LIN {X 0,Y 240.088,Z 926.359,A -85,B 0,C 180,E1 -19178.416,E2 -19178.416} C_VEL
LIN {X 0,Y 240.831,Z 922.84,A -85,B 0,C 180,E1 -19181.787,E2 -19181.787} C_VEL
LIN {X 0,Y 242.351,Z 917.839,A -85,B 0,C 180,E1 -19185.129,E2 -19185.129} C_VEL
LIN {X 0,Y 243.941,Z 913.085,A -85,B 0,C 180,E1 -19187.584,E2 -19187.584} C_VEL
LIN {X 0,Y 246.126,Z 906.104,A -85,B 0,C 180,E1 -19190.475,E2 -19190.475} C_VEL
LIN {X 0,Y 249.078,Z 897.538,A -85,B 0,C 180,E1 -19193.267,E2 -19193.267} C_VEL
LIN {X 0,Y 252.071,Z 888.617,A -85,B 0,C 180,E1 -19195.604,E2 -19195.604} C_VEL
LIN {X 0,Y 255.559,Z 877.834,A -85,B 0,C 180,E1 -19197.873,E2 -19197.873} C_VEL
LIN {X 0,Y 258.987,Z 865.759,A -85,B 0,C 180,E1 -19199.91,E2 -19199.91} C_VEL
LIN {X 0,Y 262.112,Z 853.54,A -85,B 0,C 180,E1 -19201.524,E2 -19201.524} C_VEL
LIN {X 0,Y 264.754,Z 841.815,A -85,B 0,C 180,E1 -19202.742,E2 -19202.742} C_VEL
LIN {X 0,Y 267.304,Z 827.813,A -85,B 0,C 180,E1 -19203.853,E2 -19203.853} C_VEL
LIN {X 0,Y 269.3,Z 813.813,A -85,B 0,C 180,E1 -19204.641,E2 -19204.641} C_VEL
LIN {X 0,Y 270.504,Z 800.1,A -85,B 0,C 180,E1 -19205.166,E2 -19205.166} C_VEL
LIN {X 0,Y 273.902,Z 726.368,A -85,B 0,C 180,E1 -19207.051,E2 -19207.051} C_VEL
LIN {X 0,Y 272.415,Z 716.477,A -85,B 0,C 180,E1 -19207.635,E2 -19207.635} C_VEL
LIN {X 0,Y 264.692,Z 699.058,A -85,B 0,C 180,E1 -19209.647,E2 -19209.647} C_VEL
LIN {X 0,Y 256.839,Z 683.886,A -85,B 0,C 180,E1 -19211.794,E2 -19211.794} C_VEL
LIN {X 0,Y 250.877,Z 673.683,A -85,B 0,C 180,E1 -19213.52,E2 -19213.52} C_VEL
LIN {X 0,Y 247.506,Z 668.217,A -85,B 0,C 180,E1 -19214.545,E2 -19214.545} C_VEL
LIN {X 0,Y 244.888,Z 663.741,A -85,B 0,C 180,E1 -19215.408,E2 -19215.408} C_VEL
LIN {X 0,Y 242.509,Z 656.323,A -85,B 0,C 180,E1 -19219.273,E2 -19219.273} C_VEL
LIN {X 0,Y 241.973,Z 654.468,A -85,B 0,C 180,E1 -19220.378,E2 -19220.378} C_VEL
LIN {X 0,Y 242.036,Z 654.449,A -85,B 0,C 180,E1 -19224.498,E2 -19224.498} C_VEL
LIN {X 0,Y 241.976,Z 654.432,A -85,B 0,C 180,E1 -19228.48,E2 -19228.48} C_VEL
LIN {X 0,Y 242.01,Z 654.461,A -85,B 0,C 180,E1 -19232.313,E2 -19232.313} C_VEL
LIN {X 0,Y 242.061,Z 654.455,A -85,B 0,C 180,E1 -19236.017,E2 -19236.017} C_VEL
LIN {X 0,Y 242.039,Z 654.46,A -85,B 0,C 180,E1 -19239.608,E2 -19239.608} C_VEL
LIN {X 0,Y 242.164,Z 654.443,A -85,B 0,C 180,E1 -19243.279,E2 -19243.279} C_VEL
LIN {X 0,Y 242.182,Z 654.444,A -85,B 0,C 180,E1 -19248.28,E2 -19248.28} C_VEL
LIN {X 0,Y 242.401,Z 654.404,A -85,B 0,C 180,E1 -19251.665,E2 -19251.665} C_VEL
LIN {X 0,Y 242.258,Z 654.422,A -85,B 0,C 180,E1 -19255.008,E2 -19255.008} C_VEL
LIN {X 0,Y 242.637,Z 654.387,A -85,B 0,C 180,E1 -19258.341,E2 -19258.341} C_VEL
LIN {X 0,Y 242.637,Z 654.377,A -85,B 0,C 180,E1 -19261.66,E2 -19261.66} C_VEL
LIN {X 0,Y 242.423,Z 654.403,A -85,B 0,C 180,E1 -19266.684,E2 -19266.684} C_VEL
LIN {X 0,Y 242.269,Z 654.42,A -85,B 0,C 180,E1 -19270.024,E2 -19270.024} C_VEL
LIN {X 0,Y 242.169,Z 654.432,A -85,B 0,C 180,E1 -19275.141,E2 -19275.141} C_VEL
LIN {X 0,Y 242.073,Z 654.448,A -85,B 0,C 180,E1 -19278.625,E2 -19278.625} C_VEL
LIN {X 0,Y 242.007,Z 654.463,A -85,B 0,C 180,E1 -19282.181,E2 -19282.181} C_VEL
LIN {X 0,Y 242.034,Z 654.461,A -85,B 0,C 180,E1 -19285.822,E2 -19285.822} C_VEL
LIN {X 0,Y 241.971,Z 654.433,A -85,B 0,C 180,E1 -19289.589,E2 -19289.589} C_VEL
LIN {X 0,Y 241.981,Z 654.462,A -85,B 0,C 180,E1 -19293.493,E2 -19293.493} C_VEL
LIN {X 0,Y 241.984,Z 654.464,A -85,B 0,C 180,E1 -19297.584,E2 -19297.584} C_VEL
LIN {X 0,Y 241.941,Z 654.466,A -85,B 0,C 180,E1 -19299.017,E2 -19299.017} C_VEL
LIN {X 0,Y 242.888,Z 657.248,A -85,B 0,C 180,E1 -19299.397,E2 -19299.397} C_VEL
LIN {X 0,Y 245.069,Z 659.506,A -85,B 0,C 180,E1 -19300.06,E2 -19300.06} C_VEL
LIN {X 0,Y 247.535,Z 663.319,A -85,B 0,C 180,E1 -19300.837,E2 -19300.837} C_VEL
LIN {X 0,Y 248.885,Z 665.08,A -85,B 0,C 180,E1 -19301.238,E2 -19301.238} C_VEL
LIN {X 0,Y 252.713,Z 670.642,A -85,B 0,C 180,E1 -19302.36,E2 -19302.36} C_VEL
LIN {X 0,Y 259.191,Z 680.306,A -85,B 0,C 180,E1 -19304.146,E2 -19304.146} C_VEL
LIN {X 0,Y 265.13,Z 690.246,A -85,B 0,C 180,E1 -19305.702,E2 -19305.702} C_VEL
LIN {X 0,Y 272.196,Z 704.465,A -85,B 0,C 180,E1 -19307.5,E2 -19307.5} C_VEL
LIN {X 0,Y 274.562,Z 709.751,A -85,B 0,C 180,E1 -19308.089,E2 -19308.089} C_VEL
LIN {X 0,Y 271.055,Z 786.527,A -85,B 0,C 180,E1 -19310.079,E2 -19310.079} C_VEL
LIN {X 0,Y 269.646,Z 801.309,A -85,B 0,C 180,E1 -19310.739,E2 -19310.739} C_VEL
LIN {X 0,Y 267.76,Z 814.787,A -85,B 0,C 180,E1 -19311.617,E2 -19311.617} C_VEL
LIN {X 0,Y 265.371,Z 827.421,A -85,B 0,C 180,E1 -19312.703,E2 -19312.703} C_VEL
LIN {X 0,Y 262.585,Z 840.272,A -85,B 0,C 180,E1 -19314.163,E2 -19314.163} C_VEL
LIN {X 0,Y 259.624,Z 851.868,A -85,B 0,C 180,E1 -19315.827,E2 -19315.827} C_VEL
LIN {X 0,Y 256.55,Z 862.473,A -85,B 0,C 180,E1 -19317.711,E2 -19317.711} C_VEL
LIN {X 0,Y 253.359,Z 872.972,A -85,B 0,C 180,E1 -19320.046,E2 -19320.046} C_VEL
LIN {X 0,Y 250.379,Z 881.602,A -85,B 0,C 180,E1 -19322.41,E2 -19322.41} C_VEL
LIN {X 0,Y 247.78,Z 888.746,A -85,B 0,C 180,E1 -19324.82,E2 -19324.82} C_VEL
LIN {X 0,Y 245.672,Z 894.661,A -85,B 0,C 180,E1 -19327.282,E2 -19327.282} C_VEL
LIN {X 0,Y 243.34,Z 900.946,A -85,B 0,C 180,E1 -19330.602,E2 -19330.602} C_VEL
LIN {X 0,Y 241.933,Z 904.957,A -85,B 0,C 180,E1 -19333.464,E2 -19333.464} C_VEL
LIN {X 0,Y 240.798,Z 908.016,A -85,B 0,C 180,E1 -19336.498,E2 -19336.498} C_VEL
LIN {X 0,Y 240.149,Z 910.096,A -85,B 0,C 180,E1 -19339.887,E2 -19339.887} C_VEL
LIN {X 0,Y 239.958,Z 910.837,A -85,B 0,C 180,E1 -19343.272,E2 -19343.272} C_VEL
LIN {X 0,Y 239.916,Z 910.27,A -85,B 0,C 180,E1 -19346.641,E2 -19346.641} C_VEL
LIN {X 0,Y 240.051,Z 908.394,A -85,B 0,C 180,E1 -19350,E2 -19350} C_VEL
LIN {X 0,Y 240.514,Z 905.147,A -85,B 0,C 180,E1 -19353.351,E2 -19353.351} C_VEL
LIN {X 0,Y 241.617,Z 900.424,A -85,B 0,C 180,E1 -19356.682,E2 -19356.682} C_VEL
LIN {X 0,Y 242.775,Z 895.871,A -85,B 0,C 180,E1 -19359.162,E2 -19359.162} C_VEL
LIN {X 0,Y 244.53,Z 889.16,A -85,B 0,C 180,E1 -19362.063,E2 -19362.063} C_VEL
LIN {X 0,Y 246.44,Z 881.04,A -85,B 0,C 180,E1 -19364.872,E2 -19364.872} C_VEL
LIN {X 0,Y 248.908,Z 872.445,A -85,B 0,C 180,E1 -19367.246,E2 -19367.246} C_VEL
LIN {X 0,Y 251.545,Z 862.05,A -85,B 0,C 180,E1 -19369.589,E2 -19369.589} C_VEL
LIN {X 0,Y 254.179,Z 850.427,A -85,B 0,C 180,E1 -19371.705,E2 -19371.705} C_VEL
LIN {X 0,Y 256.478,Z 838.788,A -85,B 0,C 180,E1 -19373.412,E2 -19373.412} C_VEL
LIN {X 0,Y 258.792,Z 825.949,A -85,B 0,C 180,E1 -19374.894,E2 -19374.894} C_VEL
LIN {X 0,Y 260.773,Z 812.564,A -85,B 0,C 180,E1 -19376.081,E2 -19376.081} C_VEL
LIN {X 0,Y 262.277,Z 798.574,A -85,B 0,C 180,E1 -19376.992,E2 -19376.992} C_VEL
LIN {X 0,Y 263.296,Z 784.338,A -85,B 0,C 180,E1 -19377.607,E2 -19377.607} C_VEL
LIN {X 0,Y 266.607,Z 702.616,A -85,B 0,C 180,E1 -19379.747,E2 -19379.747} C_VEL
LIN {X 0,Y 259.944,Z 686.637,A -85,B 0,C 180,E1 -19381.221,E2 -19381.221} C_VEL
LIN {X 0,Y 254.009,Z 675.196,A -85,B 0,C 180,E1 -19382.527,E2 -19382.527} C_VEL
LIN {X 0,Y 245.648,Z 661.352,A -85,B 0,C 180,E1 -19384.431,E2 -19384.431} C_VEL
LIN {X 0,Y 243.844,Z 658.424,A -85,B 0,C 180,E1 -19384.864,E2 -19384.864} C_VEL
LIN {X 0,Y 242.334,Z 655.911,A -85,B 0,C 180,E1 -19385.235,E2 -19385.235} C_VEL
LIN {X 0,Y 242,Z 654.467,A -85,B 0,C 180,E1 -19385.38,E2 -19385.38} C_VEL
LIN {X 0,Y 241.936,Z 654.453,A -85,B 0,C 180,E1 -19389.723,E2 -19389.723} C_VEL
LIN {X 0,Y 241.919,Z 654.469,A -85,B 0,C 180,E1 -19394.205,E2 -19394.205} C_VEL
LIN {X 0,Y 241.911,Z 654.475,A -85,B 0,C 180,E1 -19398.071,E2 -19398.071} C_VEL
LIN {X 0,Y 241.967,Z 654.433,A -85,B 0,C 180,E1 -19402.413,E2 -19402.413} C_VEL
LIN {X 0,Y 241.982,Z 654.466,A -85,B 0,C 180,E1 -19406.507,E2 -19406.507} C_VEL
LIN {X 0,Y 241.98,Z 654.454,A -85,B 0,C 180,E1 -19410.612,E2 -19410.612} C_VEL
LIN {X 0,Y 242.035,Z 654.455,A -85,B 0,C 180,E1 -19414.179,E2 -19414.179} C_VEL
LIN {X 0,Y 242.025,Z 654.46,A -85,B 0,C 180,E1 -19418.315,E2 -19418.315} C_VEL
LIN {X 0,Y 242.118,Z 654.43,A -85,B 0,C 180,E1 -19423.316,E2 -19423.316} C_VEL
LIN {X 0,Y 242.17,Z 654.43,A -85,B 0,C 180,E1 -19428.278,E2 -19428.278} C_VEL
LIN {X 0,Y 242.388,Z 654.408,A -85,B 0,C 180,E1 -19431.664,E2 -19431.664} C_VEL
LIN {X 0,Y 242.242,Z 654.429,A -85,B 0,C 180,E1 -19435.006,E2 -19435.006} C_VEL
LIN {X 0,Y 242.636,Z 654.386,A -85,B 0,C 180,E1 -19438.34,E2 -19438.34} C_VEL
LIN {X 0,Y 242.592,Z 654.382,A -85,B 0,C 180,E1 -19441.872,E2 -19441.872} C_VEL
LIN {X 0,Y 241.73,Z 654.5,A -85,B 0,C 180,E1 -19443.255,E2 -19443.255} C_VEL
LIN {X 0,Y 238.797,Z 654.862,A -85,B 0,C 180,E1 -19445.512,E2 -19445.512} C_VEL
LIN {X 0,Y 236.412,Z 655.16,A -85,B 0,C 180,E1 -19447.35,E2 -19447.35} C_VEL
LIN {X 0,Y 235.388,Z 655.288,A -85,B 0,C 180,E1 -19448.776,E2 -19448.776} C_VEL
LIN {X 0,Y 235.297,Z 655.295,A -85,B 0,C 180,E1 -19449.259,E2 -19449.259} C_VEL
LIN {X 0,Y 235.109,Z 655.321,A -85,B 0,C 180,E1 -19453.835,E2 -19453.835} C_VEL
LIN {X 0,Y 235.07,Z 655.326,A -85,B 0,C 180,E1 -19457.396,E2 -19457.396} C_VEL
LIN {X 0,Y 234.979,Z 655.338,A -85,B 0,C 180,E1 -19462,E2 -19462} C_VEL
LIN {X 0,Y 234.97,Z 655.334,A -85,B 0,C 180,E1 -19466.657,E2 -19466.657} C_VEL
LIN {X 0,Y 234.934,Z 655.34,A -85,B 0,C 180,E1 -19470.567,E2 -19470.567} C_VEL
LIN {X 0,Y 234.962,Z 655.339,A -85,B 0,C 180,E1 -19474.632,E2 -19474.632} C_VEL
LIN {X 0,Y 234.968,Z 655.339,A -85,B 0,C 180,E1 -19478.952,E2 -19478.952} C_VEL
LIN {X 0,Y 234.949,Z 655.341,A -85,B 0,C 180,E1 -19483.471,E2 -19483.471} C_VEL
LIN {X 0,Y 234.953,Z 655.525,A -85,B 0,C 180,E1 -19484.67,E2 -19484.67} C_VEL
LIN {X 0,Y 237.458,Z 664.503,A -85,B 0,C 180,E1 -19488.654,E2 -19488.654} C_VEL
LIN {X 0,Y 244.776,Z 678.336,A -85,B 0,C 180,E1 -19490.52,E2 -19490.52} C_VEL
LIN {X 0,Y 252.132,Z 694.464,A -85,B 0,C 180,E1 -19492.323,E2 -19492.323} C_VEL
LIN {X 0,Y 257.755,Z 708.307,A -85,B 0,C 180,E1 -19493.657,E2 -19493.657} C_VEL
LIN {X 0,Y 259.899,Z 725.152,A -85,B 0,C 180,E1 -19494.519,E2 -19494.519} C_VEL
LIN {X 0,Y 256.62,Z 803.382,A -85,B 0,C 180,E1 -19496.625,E2 -19496.625} C_VEL
LIN {X 0,Y 255.268,Z 817.931,A -85,B 0,C 180,E1 -19497.295,E2 -19497.295} C_VEL
LIN {X 0,Y 253.467,Z 831.442,A -85,B 0,C 180,E1 -19498.209,E2 -19498.209} C_VEL
LIN {X 0,Y 251.375,Z 843.741,A -85,B 0,C 180,E1 -19499.32,E2 -19499.32} C_VEL
LIN {X 0,Y 248.825,Z 856.669,A -85,B 0,C 180,E1 -19500.842,E2 -19500.842} C_VEL
LIN {X 0,Y 246.309,Z 868.123,A -85,B 0,C 180,E1 -19502.549,E2 -19502.549} C_VEL
LIN {X 0,Y 243.841,Z 878.189,A -85,B 0,C 180,E1 -19504.384,E2 -19504.384} C_VEL
LIN {X 0,Y 241.346,Z 887.356,A -85,B 0,C 180,E1 -19506.397,E2 -19506.397} C_VEL
LIN {X 0,Y 238.958,Z 896.569,A -85,B 0,C 180,E1 -19508.882,E2 -19508.882} C_VEL
LIN {X 0,Y 236.842,Z 904.466,A -85,B 0,C 180,E1 -19511.489,E2 -19511.489} C_VEL
LIN {X 0,Y 235.207,Z 911.563,A -85,B 0,C 180,E1 -19514.4,E2 -19514.4} C_VEL
LIN {X 0,Y 234.076,Z 916.69,A -85,B 0,C 180,E1 -19516.986,E2 -19516.986} C_VEL
LIN {X 0,Y 233.168,Z 921.968,A -85,B 0,C 180,E1 -19520.457,E2 -19520.457} C_VEL
LIN {X 0,Y 232.856,Z 924.929,A -85,B 0,C 180,E1 -19523.066,E2 -19523.066} C_VEL
LIN {X 0,Y 232.831,Z 926.555,A -85,B 0,C 180,E1 -19524.939,E2 -19524.939} C_VEL
LIN {X 0,Y 232.827,Z 928.419,A -85,B 0,C 180,E1 -19528.27,E2 -19528.27} C_VEL
LIN {X 0,Y 232.888,Z 928.888,A -85,B 0,C 180,E1 -19530,E2 -19530} C_VEL
LIN {X 0,Y 232.816,Z 929.01,A -85,B 0,C 180,E1 -19531.73,E2 -19531.73} C_VEL
LIN {X 0,Y 232.742,Z 928.246,A -85,B 0,C 180,E1 -19535.197,E2 -19535.197} C_VEL
LIN {X 0,Y 233.039,Z 926.14,A -85,B 0,C 180,E1 -19538.673,E2 -19538.673} C_VEL
LIN {X 0,Y 233.826,Z 922.646,A -85,B 0,C 180,E1 -19542.145,E2 -19542.145} C_VEL
LIN {X 0,Y 235.44,Z 917.672,A -85,B 0,C 180,E1 -19545.584,E2 -19545.584} C_VEL
LIN {X 0,Y 237.262,Z 912.366,A -85,B 0,C 180,E1 -19548.38,E2 -19548.38} C_VEL
LIN {X 0,Y 239.846,Z 904.878,A -85,B 0,C 180,E1 -19551.486,E2 -19551.486} C_VEL
LIN {X 0,Y 243.033,Z 896.111,A -85,B 0,C 180,E1 -19554.335,E2 -19554.335} C_VEL
LIN {X 0,Y 246.281,Z 886.961,A -85,B 0,C 180,E1 -19556.708,E2 -19556.708} C_VEL
LIN {X 0,Y 249.773,Z 876.499,A -85,B 0,C 180,E1 -19558.897,E2 -19558.897} C_VEL
LIN {X 0,Y 252.838,Z 865.845,A -85,B 0,C 180,E1 -19560.714,E2 -19560.714} C_VEL
LIN {X 0,Y 256.085,Z 853.738,A -85,B 0,C 180,E1 -19562.354,E2 -19562.354} C_VEL
LIN {X 0,Y 258.826,Z 842.104,A -85,B 0,C 180,E1 -19563.59,E2 -19563.59} C_VEL
LIN {X 0,Y 261.467,Z 828.337,A -85,B 0,C 180,E1 -19564.715,E2 -19564.715} C_VEL
LIN {X 0,Y 263.632,Z 813.751,A -85,B 0,C 180,E1 -19565.555,E2 -19565.555} C_VEL
LIN {X 0,Y 264.913,Z 799.46,A -85,B 0,C 180,E1 -19566.11,E2 -19566.11} C_VEL
LIN {X 0,Y 268.353,Z 727.432,A -85,B 0,C 180,E1 -19567.979,E2 -19567.979} C_VEL
LIN {X 0,Y 267.061,Z 719.125,A -85,B 0,C 180,E1 -19568.499,E2 -19568.499} C_VEL
LIN {X 0,Y 259.143,Z 701.17,A -85,B 0,C 180,E1 -19570.667,E2 -19570.667} C_VEL
LIN {X 0,Y 251.705,Z 687.021,A -85,B 0,C 180,E1 -19572.8,E2 -19572.8} C_VEL
LIN {X 0,Y 246.944,Z 678.673,A -85,B 0,C 180,E1 -19574.25,E2 -19574.25} C_VEL
LIN {X 0,Y 240.455,Z 668.201,A -85,B 0,C 180,E1 -19576.349,E2 -19576.349} C_VEL
LIN {X 0,Y 237.454,Z 663.229,A -85,B 0,C 180,E1 -19577.462,E2 -19577.462} C_VEL
LIN {X 0,Y 234.985,Z 655.315,A -85,B 0,C 180,E1 -19581.981,E2 -19581.981} C_VEL
LIN {X 0,Y 234.95,Z 655.32,A -85,B 0,C 180,E1 -19586.883,E2 -19586.883} C_VEL
LIN {X 0,Y 234.954,Z 655.339,A -85,B 0,C 180,E1 -19591.407,E2 -19591.407} C_VEL
LIN {X 0,Y 234.99,Z 655.336,A -85,B 0,C 180,E1 -19595.247,E2 -19595.247} C_VEL
LIN {X 0,Y 235.012,Z 655.332,A -85,B 0,C 180,E1 -19598.97,E2 -19598.97} C_VEL
LIN {X 0,Y 235.097,Z 655.32,A -85,B 0,C 180,E1 -19603.06,E2 -19603.06} C_VEL
LIN {X 0,Y 235.115,Z 655.32,A -85,B 0,C 180,E1 -19607.923,E2 -19607.923} C_VEL
LIN {X 0,Y 235.332,Z 655.283,A -85,B 0,C 180,E1 -19611.413,E2 -19611.413} C_VEL
LIN {X 0,Y 235.394,Z 655.289,A -85,B 0,C 180,E1 -19613.142,E2 -19613.142} C_VEL
LIN {X 0,Y 235.597,Z 655.265,A -85,B 0,C 180,E1 -19618.291,E2 -19618.291} C_VEL
LIN {X 0,Y 235.597,Z 655.254,A -85,B 0,C 180,E1 -19621.71,E2 -19621.71} C_VEL
LIN {X 0,Y 235.375,Z 655.283,A -85,B 0,C 180,E1 -19626.86,E2 -19626.86} C_VEL
LIN {X 0,Y 235.216,Z 655.297,A -85,B 0,C 180,E1 -19630.328,E2 -19630.328} C_VEL
LIN {X 0,Y 235.115,Z 655.312,A -85,B 0,C 180,E1 -19635.607,E2 -19635.607} C_VEL
LIN {X 0,Y 235.009,Z 655.325,A -85,B 0,C 180,E1 -19639.206,E2 -19639.206} C_VEL
LIN {X 0,Y 234.952,Z 655.335,A -85,B 0,C 180,E1 -19642.884,E2 -19642.884} C_VEL
LIN {X 0,Y 234.948,Z 655.332,A -85,B 0,C 180,E1 -19646.661,E2 -19646.661} C_VEL
LIN {X 0,Y 234.901,Z 655.321,A -85,B 0,C 180,E1 -19650.573,E2 -19650.573} C_VEL
LIN {X 0,Y 234.927,Z 655.341,A -85,B 0,C 180,E1 -19654.639,E2 -19654.639} C_VEL
LIN {X 0,Y 234.918,Z 655.376,A -85,B 0,C 180,E1 -19657.087,E2 -19657.087} C_VEL
LIN {X 0,Y 235.79,Z 657.948,A -85,B 0,C 180,E1 -19657.463,E2 -19657.463} C_VEL
LIN {X 0,Y 237.848,Z 660.234,A -85,B 0,C 180,E1 -19658.157,E2 -19658.157} C_VEL
LIN {X 0,Y 238.51,Z 661.013,A -85,B 0,C 180,E1 -19658.377,E2 -19658.377} C_VEL
LIN {X 0,Y 240.624,Z 664.296,A -85,B 0,C 180,E1 -19659.102,E2 -19659.102} C_VEL
LIN {X 0,Y 242.07,Z 666.019,A -85,B 0,C 180,E1 -19659.563,E2 -19659.563} C_VEL
LIN {X 0,Y 250.555,Z 678.145,A -85,B 0,C 180,E1 -19662.162,E2 -19662.162} C_VEL
LIN {X 0,Y 259.292,Z 692.068,A -85,B 0,C 180,E1 -19664.605,E2 -19664.605} C_VEL
LIN {X 0,Y 267.106,Z 707.667,A -85,B 0,C 180,E1 -19666.69,E2 -19666.69} C_VEL
LIN {X 0,Y 268.933,Z 711.817,A -85,B 0,C 180,E1 -19667.168,E2 -19667.168} C_VEL
LIN {X 0,Y 267.067,Z 753.218,A -85,B 0,C 180,E1 -19668.251,E2 -19668.251} C_VEL
LIN {X 0,Y 265.399,Z 787.321,A -85,B 0,C 180,E1 -19669.175,E2 -19669.175} C_VEL
LIN {X 0,Y 263.941,Z 801.924,A -85,B 0,C 180,E1 -19669.844,E2 -19669.844} C_VEL
LIN {X 0,Y 261.893,Z 815.882,A -85,B 0,C 180,E1 -19670.779,E2 -19670.779} C_VEL
LIN {X 0,Y 259.484,Z 828.085,A -85,B 0,C 180,E1 -19671.857,E2 -19671.857} C_VEL
LIN {X 0,Y 256.459,Z 841.42,A -85,B 0,C 180,E1 -19673.414,E2 -19673.414} C_VEL
LIN {X 0,Y 253.39,Z 852.858,A -85,B 0,C 180,E1 -19675.107,E2 -19675.107} C_VEL
LIN {X 0,Y 250.494,Z 862.361,A -85,B 0,C 180,E1 -19676.832,E2 -19676.832} C_VEL
LIN {X 0,Y 247.159,Z 872.924,A -85,B 0,C 180,E1 -19679.214,E2 -19679.214} C_VEL
LIN {X 0,Y 244.011,Z 881.608,A -85,B 0,C 180,E1 -19681.626,E2 -19681.626} C_VEL
LIN {X 0,Y 240.87,Z 889.951,A -85,B 0,C 180,E1 -19684.53,E2 -19684.53} C_VEL
LIN {X 0,Y 238.345,Z 896.529,A -85,B 0,C 180,E1 -19687.46,E2 -19687.46} C_VEL
LIN {X 0,Y 236.048,Z 902.381,A -85,B 0,C 180,E1 -19690.882,E2 -19690.882} C_VEL
LIN {X 0,Y 234.444,Z 906.642,A -85,B 0,C 180,E1 -19694.348,E2 -19694.348} C_VEL
LIN {X 0,Y 233.344,Z 909.448,A -85,B 0,C 180,E1 -19697.829,E2 -19697.829} C_VEL
LIN {X 0,Y 232.919,Z 910.883,A -85,B 0,C 180,E1 -19701.323,E2 -19701.323} C_VEL
LIN {X 0,Y 232.848,Z 910.997,A -85,B 0,C 180,E1 -19704.805,E2 -19704.805} C_VEL
LIN {X 0,Y 232.898,Z 909.81,A -85,B 0,C 180,E1 -19708.271,E2 -19708.271} C_VEL
LIN {X 0,Y 233.148,Z 907.301,A -85,B 0,C 180,E1 -19711.728,E2 -19711.728} C_VEL
LIN {X 0,Y 233.95,Z 903.37,A -85,B 0,C 180,E1 -19715.171,E2 -19715.171} C_VEL
LIN {X 0,Y 235.4,Z 897.898,A -85,B 0,C 180,E1 -19718.585,E2 -19718.585} C_VEL
LIN {X 0,Y 236.816,Z 892.722,A -85,B 0,C 180,E1 -19721.122,E2 -19721.122} C_VEL
LIN {X 0,Y 238.671,Z 885.274,A -85,B 0,C 180,E1 -19724.06,E2 -19724.06} C_VEL
LIN {X 0,Y 240.88,Z 877.503,A -85,B 0,C 180,E1 -19726.527,E2 -19726.527} C_VEL
LIN {X 0,Y 243.5,Z 868.124,A -85,B 0,C 180,E1 -19728.948,E2 -19728.948} C_VEL
LIN {X 0,Y 246.133,Z 857.752,A -85,B 0,C 180,E1 -19731.131,E2 -19731.131} C_VEL
LIN {X 0,Y 248.41,Z 847.594,A -85,B 0,C 180,E1 -19732.893,E2 -19732.893} C_VEL
LIN {X 0,Y 250.613,Z 836.757,A -85,B 0,C 180,E1 -19734.434,E2 -19734.434} C_VEL
LIN {X 0,Y 252.718,Z 825.153,A -85,B 0,C 180,E1 -19735.755,E2 -19735.755} C_VEL
LIN {X 0,Y 254.793,Z 811.326,A -85,B 0,C 180,E1 -19736.962,E2 -19736.962} C_VEL
LIN {X 0,Y 256.248,Z 797.577,A -85,B 0,C 180,E1 -19737.846,E2 -19737.846} C_VEL
LIN {X 0,Y 257.269,Z 783.689,A -85,B 0,C 180,E1 -19738.433,E2 -19738.433} C_VEL
LIN {X 0,Y 260.523,Z 704.324,A -85,B 0,C 180,E1 -19740.558,E2 -19740.558} C_VEL
LIN {X 0,Y 253.921,Z 688.54,A -85,B 0,C 180,E1 -19742.087,E2 -19742.087} C_VEL
LIN {X 0,Y 246.236,Z 674.417,A -85,B 0,C 180,E1 -19743.858,E2 -19743.858} C_VEL
LIN {X 0,Y 238.878,Z 662.529,A -85,B 0,C 180,E1 -19745.641,E2 -19745.641} C_VEL
LIN {X 0,Y 237.106,Z 659.66,A -85,B 0,C 180,E1 -19746.094,E2 -19746.094} C_VEL
LIN {X 0,Y 235.318,Z 657.035,A -85,B 0,C 180,E1 -19746.55,E2 -19746.55} C_VEL
LIN {X 0,Y 234.909,Z 655.347,A -85,B 0,C 180,E1 -19746.753,E2 -19746.753} C_VEL
LIN {X 0,Y 234.915,Z 655.332,A -85,B 0,C 180,E1 -19748.935,E2 -19748.935} C_VEL
LIN {X 0,Y 234.878,Z 655.347,A -85,B 0,C 180,E1 -19753.489,E2 -19753.489} C_VEL
LIN {X 0,Y 234.865,Z 655.35,A -85,B 0,C 180,E1 -19756.508,E2 -19756.508} C_VEL
LIN {X 0,Y 234.92,Z 655.323,A -85,B 0,C 180,E1 -19761.078,E2 -19761.078} C_VEL
LIN {X 0,Y 234.924,Z 655.335,A -85,B 0,C 180,E1 -19765.36,E2 -19765.36} C_VEL
LIN {X 0,Y 234.902,Z 655.333,A -85,B 0,C 180,E1 -19769.427,E2 -19769.427} C_VEL
LIN {X 0,Y 234.971,Z 655.336,A -85,B 0,C 180,E1 -19773.806,E2 -19773.806} C_VEL
LIN {X 0,Y 234.992,Z 655.338,A -85,B 0,C 180,E1 -19778.967,E2 -19778.967} C_VEL
LIN {X 0,Y 235.059,Z 655.307,A -85,B 0,C 180,E1 -19783.092,E2 -19783.092} C_VEL
LIN {X 0,Y 235.102,Z 655.313,A -85,B 0,C 180,E1 -19787.921,E2 -19787.921} C_VEL
LIN {X 0,Y 235.322,Z 655.286,A -85,B 0,C 180,E1 -19791.412,E2 -19791.412} C_VEL
LIN {X 0,Y 235.358,Z 655.292,A -85,B 0,C 180,E1 -19793.139,E2 -19793.139} C_VEL
LIN {X 0,Y 235.595,Z 655.263,A -85,B 0,C 180,E1 -19798.29,E2 -19798.29} C_VEL
LIN {X 0,Y 235.581,Z 655.256,A -85,B 0,C 180,E1 -19801.781,E2 -19801.781} C_VEL
LIN {X 0,Y 235.375,Z 655.285,A -85,B 0,C 180,E1 -19806.859,E2 -19806.859} C_VEL
LIN {X 0,Y 235.297,Z 655.295,A -85,B 0,C 180,E1 -19809.259,E2 -19809.259} C_VEL
LIN {X 0,Y 234.588,Z 655.383,A -85,B 0,C 180,E1 -19810.687,E2 -19810.687} C_VEL
LIN {X 0,Y 231.655,Z 655.753,A -85,B 0,C 180,E1 -19813.013,E2 -19813.013} C_VEL
LIN {X 0,Y 229.179,Z 656.054,A -85,B 0,C 180,E1 -19814.91,E2 -19814.91} C_VEL
LIN {X 0,Y 228.12,Z 656.187,A -85,B 0,C 180,E1 -19816.385,E2 -19816.385} C_VEL
LIN {X 0,Y 228.035,Z 656.199,A -85,B 0,C 180,E1 -19816.885,E2 -19816.885} C_VEL
LIN {X 0,Y 227.949,Z 656.213,A -85,B 0,C 180,E1 -19821.714,E2 -19821.714} C_VEL
LIN {X 0,Y 227.944,Z 656.21,A -85,B 0,C 180,E1 -19826.602,E2 -19826.602} C_VEL
LIN {X 0,Y 227.91,Z 656.215,A -85,B 0,C 180,E1 -19830.296,E2 -19830.296} C_VEL
LIN {X 0,Y 227.891,Z 656.219,A -85,B 0,C 180,E1 -19833.718,E2 -19833.718} C_VEL
LIN {X 0,Y 227.872,Z 656.226,A -85,B 0,C 180,E1 -19838.085,E2 -19838.085} C_VEL
LIN {X 0,Y 227.895,Z 656.221,A -85,B 0,C 180,E1 -19842.722,E2 -19842.722} C_VEL
LIN {X 0,Y 227.914,Z 656.299,A -85,B 0,C 180,E1 -19843.474,E2 -19843.474} C_VEL
LIN {X 0,Y 230.089,Z 664.076,A -85,B 0,C 180,E1 -19847.144,E2 -19847.144} C_VEL
LIN {X 0,Y 232.529,Z 668.575,A -85,B 0,C 180,E1 -19847.83,E2 -19847.83} C_VEL
LIN {X 0,Y 238.864,Z 680.448,A -85,B 0,C 180,E1 -19849.524,E2 -19849.524} C_VEL
LIN {X 0,Y 246.196,Z 696.303,A -85,B 0,C 180,E1 -19851.407,E2 -19851.407} C_VEL
LIN {X 0,Y 252.056,Z 710.872,A -85,B 0,C 180,E1 -19852.87,E2 -19852.87} C_VEL
LIN {X 0,Y 253.95,Z 726.459,A -85,B 0,C 180,E1 -19853.686,E2 -19853.686} C_VEL
LIN {X 0,Y 250.594,Z 802.921,A -85,B 0,C 180,E1 -19855.778,E2 -19855.778} C_VEL
LIN {X 0,Y 249.212,Z 817.485,A -85,B 0,C 180,E1 -19856.457,E2 -19856.457} C_VEL
LIN {X 0,Y 247.489,Z 830.481,A -85,B 0,C 180,E1 -19857.347,E2 -19857.347} C_VEL
LIN {X 0,Y 245.274,Z 842.926,A -85,B 0,C 180,E1 -19858.471,E2 -19858.471} C_VEL
LIN {X 0,Y 242.609,Z 855.956,A -85,B 0,C 180,E1 -19860.019,E2 -19860.019} C_VEL
LIN {X 0,Y 240.103,Z 867.049,A -85,B 0,C 180,E1 -19861.688,E2 -19861.688} C_VEL
LIN {X 0,Y 237.72,Z 876.634,A -85,B 0,C 180,E1 -19863.438,E2 -19863.438} C_VEL
LIN {X 0,Y 234.797,Z 886.831,A -85,B 0,C 180,E1 -19865.696,E2 -19865.696} C_VEL
LIN {X 0,Y 232.288,Z 896.086,A -85,B 0,C 180,E1 -19868.245,E2 -19868.245} C_VEL
LIN {X 0,Y 229.775,Z 904.979,A -85,B 0,C 180,E1 -19871.292,E2 -19871.292} C_VEL
LIN {X 0,Y 228.323,Z 911.149,A -85,B 0,C 180,E1 -19873.917,E2 -19873.917} C_VEL
LIN {X 0,Y 227.098,Z 916.3,A -85,B 0,C 180,E1 -19876.579,E2 -19876.579} C_VEL
LIN {X 0,Y 226.124,Z 921.612,A -85,B 0,C 180,E1 -19880.157,E2 -19880.157} C_VEL
LIN {X 0,Y 225.788,Z 924.587,A -85,B 0,C 180,E1 -19882.848,E2 -19882.848} C_VEL
LIN {X 0,Y 225.718,Z 926.452,A -85,B 0,C 180,E1 -19885.106,E2 -19885.106} C_VEL
LIN {X 0,Y 225.738,Z 928.121,A -85,B 0,C 180,E1 -19888.216,E2 -19888.216} C_VEL
LIN {X 0,Y 225.82,Z 928.605,A -85,B 0,C 180,E1 -19890,E2 -19890} C_VEL
LIN {X 0,Y 225.726,Z 928.741,A -85,B 0,C 180,E1 -19891.784,E2 -19891.784} C_VEL
LIN {X 0,Y 225.648,Z 928.002,A -85,B 0,C 180,E1 -19895.361,E2 -19895.361} C_VEL
LIN {X 0,Y 225.984,Z 925.92,A -85,B 0,C 180,E1 -19898.946,E2 -19898.946} C_VEL
LIN {X 0,Y 226.837,Z 922.451,A -85,B 0,C 180,E1 -19902.526,E2 -19902.526} C_VEL
LIN {X 0,Y 228.55,Z 917.505,A -85,B 0,C 180,E1 -19906.066,E2 -19906.066} C_VEL
LIN {X 0,Y 230.559,Z 911.902,A -85,B 0,C 180,E1 -19909.1,E2 -19909.1} C_VEL
LIN {X 0,Y 233.221,Z 904.773,A -85,B 0,C 180,E1 -19912.128,E2 -19912.128} C_VEL
LIN {X 0,Y 236.528,Z 896.044,A -85,B 0,C 180,E1 -19915.05,E2 -19915.05} C_VEL
LIN {X 0,Y 239.952,Z 886.937,A -85,B 0,C 180,E1 -19917.471,E2 -19917.471} C_VEL
LIN {X 0,Y 243.534,Z 876.651,A -85,B 0,C 180,E1 -19919.68,E2 -19919.68} C_VEL
LIN {X 0,Y 246.764,Z 865.934,A -85,B 0,C 180,E1 -19921.556,E2 -19921.556} C_VEL
LIN {X 0,Y 250.139,Z 853.919,A -85,B 0,C 180,E1 -19923.222,E2 -19923.222} C_VEL
LIN {X 0,Y 252.947,Z 842.378,A -85,B 0,C 180,E1 -19924.479,E2 -19924.479} C_VEL
LIN {X 0,Y 255.695,Z 828.841,A -85,B 0,C 180,E1 -19925.616,E2 -19925.616} C_VEL
LIN {X 0,Y 257.911,Z 814.608,A -85,B 0,C 180,E1 -19926.469,E2 -19926.469} C_VEL
LIN {X 0,Y 259.333,Z 799.984,A -85,B 0,C 180,E1 -19927.057,E2 -19927.057} C_VEL
LIN {X 0,Y 262.904,Z 728.582,A -85,B 0,C 180,E1 -19928.939,E2 -19928.939} C_VEL
LIN {X 0,Y 261.92,Z 722.056,A -85,B 0,C 180,E1 -19929.359,E2 -19929.359} C_VEL
LIN {X 0,Y 254.566,Z 705.304,A -85,B 0,C 180,E1 -19931.465,E2 -19931.465} C_VEL
LIN {X 0,Y 247.213,Z 691,A -85,B 0,C 180,E1 -19933.681,E2 -19933.681} C_VEL
LIN {X 0,Y 242.33,Z 682.54,A -85,B 0,C 180,E1 -19935.236,E2 -19935.236} C_VEL
LIN {X 0,Y 236.819,Z 673.453,A -85,B 0,C 180,E1 -19937.109,E2 -19937.109} C_VEL
LIN {X 0,Y 233.245,Z 667.962,A -85,B 0,C 180,E1 -19938.393,E2 -19938.393} C_VEL
LIN {X 0,Y 230.312,Z 663.442,A -85,B 0,C 180,E1 -19939.505,E2 -19939.505} C_VEL
LIN {X 0,Y 230.03,Z 662.822,A -85,B 0,C 180,E1 -19939.675,E2 -19939.675} C_VEL
LIN {X 0,Y 228.788,Z 658.767,A -85,B 0,C 180,E1 -19942.094,E2 -19942.094} C_VEL
LIN {X 0,Y 227.923,Z 656.197,A -85,B 0,C 180,E1 -19943.796,E2 -19943.796} C_VEL
LIN {X 0,Y 227.873,Z 656.188,A -85,B 0,C 180,E1 -19948.379,E2 -19948.379} C_VEL
LIN {X 0,Y 227.887,Z 656.219,A -85,B 0,C 180,E1 -19952.446,E2 -19952.446} C_VEL
LIN {X 0,Y 227.916,Z 656.214,A -85,B 0,C 180,E1 -19956.368,E2 -19956.368} C_VEL
LIN {X 0,Y 227.944,Z 656.214,A -85,B 0,C 180,E1 -19960.175,E2 -19960.175} C_VEL
LIN {X 0,Y 228.058,Z 656.203,A -85,B 0,C 180,E1 -19963.898,E2 -19963.898} C_VEL
LIN {X 0,Y 228.073,Z 656.194,A -85,B 0,C 180,E1 -19967.544,E2 -19967.544} C_VEL
LIN {X 0,Y 228.268,Z 656.162,A -85,B 0,C 180,E1 -19971.145,E2 -19971.145} C_VEL
LIN {X 0,Y 228.341,Z 656.168,A -85,B 0,C 180,E1 -19972.929,E2 -19972.929} C_VEL
LIN {X 0,Y 228.555,Z 656.142,A -85,B 0,C 180,E1 -19978.238,E2 -19978.238} C_VEL
LIN {X 0,Y 228.556,Z 656.131,A -85,B 0,C 180,E1 -19981.763,E2 -19981.763} C_VEL
LIN {X 0,Y 228.326,Z 656.163,A -85,B 0,C 180,E1 -19987.073,E2 -19987.073} C_VEL
LIN {X 0,Y 228.147,Z 656.178,A -85,B 0,C 180,E1 -19990.652,E2 -19990.652} C_VEL
LIN {X 0,Y 228.067,Z 656.191,A -85,B 0,C 180,E1 -19994.273,E2 -19994.273} C_VEL
LIN {X 0,Y 228.004,Z 656.206,A -85,B 0,C 180,E1 -19997.954,E2 -19997.954} C_VEL
LIN {X 0,Y 227.925,Z 656.214,A -85,B 0,C 180,E1 -20002.325,E2 -20002.325} C_VEL
LIN {X 0,Y 227.924,Z 656.207,A -85,B 0,C 180,E1 -20006.593,E2 -20006.593} C_VEL
LIN {X 0,Y 227.875,Z 656.192,A -85,B 0,C 180,E1 -20010.281,E2 -20010.281} C_VEL
LIN {X 0,Y 227.87,Z 656.225,A -85,B 0,C 180,E1 -20014.926,E2 -20014.926} C_VEL
LIN {X 0,Y 228.687,Z 658.746,A -85,B 0,C 180,E1 -20015.321,E2 -20015.321} C_VEL
LIN {X 0,Y 230.6,Z 660.958,A -85,B 0,C 180,E1 -20016.041,E2 -20016.041} C_VEL
LIN {X 0,Y 231.645,Z 661.957,A -85,B 0,C 180,E1 -20016.414,E2 -20016.414} C_VEL
LIN {X 0,Y 233.781,Z 665.214,A -85,B 0,C 180,E1 -20017.214,E2 -20017.214} C_VEL
LIN {X 0,Y 235.338,Z 667.108,A -85,B 0,C 180,E1 -20017.758,E2 -20017.758} C_VEL
LIN {X 0,Y 238.1,Z 670.794,A -85,B 0,C 180,E1 -20018.705,E2 -20018.705} C_VEL
LIN {X 0,Y 247.138,Z 684.018,A -85,B 0,C 180,E1 -20021.594,E2 -20021.594} C_VEL
LIN {X 0,Y 255.317,Z 697.281,A -85,B 0,C 180,E1 -20023.968,E2 -20023.968} C_VEL
LIN {X 0,Y 262.377,Z 711.705,A -85,B 0,C 180,E1 -20025.937,E2 -20025.937} C_VEL
LIN {X 0,Y 263.516,Z 714.232,A -85,B 0,C 180,E1 -20026.246,E2 -20026.246} C_VEL
LIN {X 0,Y 259.915,Z 786.932,A -85,B 0,C 180,E1 -20028.188,E2 -20028.188} C_VEL
LIN {X 0,Y 258.495,Z 800.999,A -85,B 0,C 180,E1 -20028.817,E2 -20028.817} C_VEL
LIN {X 0,Y 256.382,Z 815.269,A -85,B 0,C 180,E1 -20029.767,E2 -20029.767} C_VEL
LIN {X 0,Y 254.031,Z 826.894,A -85,B 0,C 180,E1 -20030.774,E2 -20030.774} C_VEL
LIN {X 0,Y 251.123,Z 839.702,A -85,B 0,C 180,E1 -20032.251,E2 -20032.251} C_VEL
LIN {X 0,Y 247.84,Z 851.492,A -85,B 0,C 180,E1 -20033.956,E2 -20033.956} C_VEL
LIN {X 0,Y 244.514,Z 862.253,A -85,B 0,C 180,E1 -20035.911,E2 -20035.911} C_VEL
LIN {X 0,Y 241.621,Z 871.102,A -85,B 0,C 180,E1 -20037.894,E2 -20037.894} C_VEL
LIN {X 0,Y 238.222,Z 880.261,A -85,B 0,C 180,E1 -20040.386,E2 -20040.386} C_VEL
LIN {X 0,Y 234.805,Z 888.856,A -85,B 0,C 180,E1 -20043.323,E2 -20043.323} C_VEL
LIN {X 0,Y 232.413,Z 894.854,A -85,B 0,C 180,E1 -20045.906,E2 -20045.906} C_VEL
LIN {X 0,Y 229.796,Z 901.216,A -85,B 0,C 180,E1 -20049.408,E2 -20049.408} C_VEL
LIN {X 0,Y 227.993,Z 905.802,A -85,B 0,C 180,E1 -20052.863,E2 -20052.863} C_VEL
LIN {X 0,Y 226.878,Z 908.424,A -85,B 0,C 180,E1 -20055.652,E2 -20055.652} C_VEL
LIN {X 0,Y 226.034,Z 910.568,A -85,B 0,C 180,E1 -20059.248,E2 -20059.248} C_VEL
LIN {X 0,Y 225.789,Z 911.369,A -85,B 0,C 180,E1 -20062.848,E2 -20062.848} C_VEL
LIN {X 0,Y 225.764,Z 911.244,A -85,B 0,C 180,E1 -20064.984,E2 -20064.984} C_VEL
LIN {X 0,Y 225.805,Z 910.122,A -85,B 0,C 180,E1 -20068.217,E2 -20068.217} C_VEL
LIN {X 0,Y 226.078,Z 907.65,A -85,B 0,C 180,E1 -20071.782,E2 -20071.782} C_VEL
LIN {X 0,Y 226.909,Z 903.764,A -85,B 0,C 180,E1 -20075.332,E2 -20075.332} C_VEL
LIN {X 0,Y 228.414,Z 898.328,A -85,B 0,C 180,E1 -20078.85,E2 -20078.85} C_VEL
LIN {X 0,Y 229.879,Z 893.187,A -85,B 0,C 180,E1 -20081.462,E2 -20081.462} C_VEL
LIN {X 0,Y 231.816,Z 885.787,A -85,B 0,C 180,E1 -20084.485,E2 -20084.485} C_VEL
LIN {X 0,Y 234.126,Z 878.063,A -85,B 0,C 180,E1 -20087.018,E2 -20087.018} C_VEL
LIN {X 0,Y 236.845,Z 868.743,A -85,B 0,C 180,E1 -20089.501,E2 -20089.501} C_VEL
LIN {X 0,Y 239.794,Z 857.385,A -85,B 0,C 180,E1 -20091.943,E2 -20091.943} C_VEL
LIN {X 0,Y 242.461,Z 845.812,A -85,B 0,C 180,E1 -20093.942,E2 -20093.942} C_VEL
LIN {X 0,Y 245.114,Z 832.943,A -85,B 0,C 180,E1 -20095.701,E2 -20095.701} C_VEL
LIN {X 0,Y 247.586,Z 819.305,A -85,B 0,C 180,E1 -20097.126,E2 -20097.126} C_VEL
LIN {X 0,Y 249.413,Z 805.378,A -85,B 0,C 180,E1 -20098.221,E2 -20098.221} C_VEL
LIN {X 0,Y 250.7,Z 791.699,A -85,B 0,C 180,E1 -20098.977,E2 -20098.977} C_VEL
LIN {X 0,Y 251.571,Z 776.399,A -85,B 0,C 180,E1 -20099.497,E2 -20099.497} C_VEL
LIN {X 0,Y 254.606,Z 706.354,A -85,B 0,C 180,E1 -20101.379,E2 -20101.379} C_VEL
LIN {X 0,Y 248.395,Z 691.54,A -85,B 0,C 180,E1 -20102.884,E2 -20102.884} C_VEL
LIN {X 0,Y 241.063,Z 678.151,A -85,B 0,C 180,E1 -20104.648,E2 -20104.648} C_VEL
LIN {X 0,Y 232.817,Z 664.699,A -85,B 0,C 180,E1 -20106.758,E2 -20106.758} C_VEL
LIN {X 0,Y 230.721,Z 661.477,A -85,B 0,C 180,E1 -20107.321,E2 -20107.321} C_VEL
LIN {X 0,Y 229.705,Z 660.173,A -85,B 0,C 180,E1 -20107.589,E2 -20107.589} C_VEL
LIN {X 0,Y 228.202,Z 657.762,A -85,B 0,C 180,E1 -20108.011,E2 -20108.011} C_VEL
LIN {X 0,Y 227.855,Z 656.219,A -85,B 0,C 180,E1 -20108.184,E2 -20108.184} C_VEL
LIN {X 0,Y 227.803,Z 656.234,A -85,B 0,C 180,E1 -20112.745,E2 -20112.745} C_VEL
LIN {X 0,Y 227.823,Z 656.231,A -85,B 0,C 180,E1 -20115.196,E2 -20115.196} C_VEL
LIN {X 0,Y 227.801,Z 656.232,A -85,B 0,C 180,E1 -20119.617,E2 -20119.617} C_VEL
LIN {X 0,Y 227.864,Z 656.195,A -85,B 0,C 180,E1 -20124.124,E2 -20124.124} C_VEL
LIN {X 0,Y 227.859,Z 656.219,A -85,B 0,C 180,E1 -20128.375,E2 -20128.375} C_VEL
LIN {X 0,Y 227.858,Z 656.226,A -85,B 0,C 180,E1 -20132.441,E2 -20132.441} C_VEL
LIN {X 0,Y 227.896,Z 656.203,A -85,B 0,C 180,E1 -20136.365,E2 -20136.365} C_VEL
LIN {X 0,Y 227.927,Z 656.214,A -85,B 0,C 180,E1 -20140.173,E2 -20140.173} C_VEL
LIN {X 0,Y 228.027,Z 656.189,A -85,B 0,C 180,E1 -20143.895,E2 -20143.895} C_VEL
LIN {X 0,Y 228.06,Z 656.193,A -85,B 0,C 180,E1 -20147.542,E2 -20147.542} C_VEL
LIN {X 0,Y 228.26,Z 656.163,A -85,B 0,C 180,E1 -20151.144,E2 -20151.144} C_VEL
LIN {X 0,Y 228.31,Z 656.17,A -85,B 0,C 180,E1 -20152.927,E2 -20152.927} C_VEL
LIN {X 0,Y 228.553,Z 656.141,A -85,B 0,C 180,E1 -20158.237,E2 -20158.237} C_VEL
LIN {X 0,Y 228.556,Z 656.131,A -85,B 0,C 180,E1 -20161.762,E2 -20161.762} C_VEL
LIN {X 0,Y 228.326,Z 656.164,A -85,B 0,C 180,E1 -20167.072,E2 -20167.072} C_VEL
LIN {X 0,Y 228.148,Z 656.18,A -85,B 0,C 180,E1 -20170.651,E2 -20170.651} C_VEL
LIN {X 0,Y 228.067,Z 656.194,A -85,B 0,C 180,E1 -20174.271,E2 -20174.271} C_VEL
LIN {X 0,Y 228.035,Z 656.199,A -85,B 0,C 180,E1 -20176.885,E2 -20176.885} C_VEL
LIN {X 0,Y 227.363,Z 656.291,A -85,B 0,C 180,E1 -20178.358,E2 -20178.358} C_VEL
LIN {X 0,Y 224.483,Z 656.653,A -85,B 0,C 180,E1 -20180.759,E2 -20180.759} C_VEL
LIN {X 0,Y 222.02,Z 656.954,A -85,B 0,C 180,E1 -20182.718,E2 -20182.718} C_VEL
LIN {X 0,Y 220.947,Z 657.08,A -85,B 0,C 180,E1 -20184.24,E2 -20184.24} C_VEL
LIN {X 0,Y 220.851,Z 657.09,A -85,B 0,C 180,E1 -20184.757,E2 -20184.757} C_VEL
LIN {X 0,Y 220.838,Z 657.097,A -85,B 0,C 180,E1 -20188.513,E2 -20188.513} C_VEL
LIN {X 0,Y 220.826,Z 657.103,A -85,B 0,C 180,E1 -20192.754,E2 -20192.754} C_VEL
LIN {X 0,Y 220.839,Z 657.098,A -85,B 0,C 180,E1 -20197.287,E2 -20197.287} C_VEL
LIN {X 0,Y 220.866,Z 657.094,A -85,B 0,C 180,E1 -20202.147,E2 -20202.147} C_VEL
LIN {X 0,Y 222.802,Z 663.92,A -85,B 0,C 180,E1 -20205.527,E2 -20205.527} C_VEL
LIN {X 0,Y 225.39,Z 668.456,A -85,B 0,C 180,E1 -20206.304,E2 -20206.304} C_VEL
LIN {X 0,Y 233.343,Z 683.131,A -85,B 0,C 180,E1 -20208.562,E2 -20208.562} C_VEL
LIN {X 0,Y 240.484,Z 698.613,A -85,B 0,C 180,E1 -20210.493,E2 -20210.493} C_VEL
LIN {X 0,Y 246.37,Z 713.317,A -85,B 0,C 180,E1 -20212.036,E2 -20212.036} C_VEL
LIN {X 0,Y 248.065,Z 727.448,A -85,B 0,C 180,E1 -20212.804,E2 -20212.804} C_VEL
LIN {X 0,Y 244.633,Z 802.226,A -85,B 0,C 180,E1 -20214.881,E2 -20214.881} C_VEL
LIN {X 0,Y 243.201,Z 817.028,A -85,B 0,C 180,E1 -20215.575,E2 -20215.575} C_VEL
LIN {X 0,Y 241.312,Z 830.638,A -85,B 0,C 180,E1 -20216.527,E2 -20216.527} C_VEL
LIN {X 0,Y 239.197,Z 842.098,A -85,B 0,C 180,E1 -20217.573,E2 -20217.573} C_VEL
LIN {X 0,Y 236.444,Z 855.237,A -85,B 0,C 180,E1 -20219.154,E2 -20219.154} C_VEL
LIN {X 0,Y 233.69,Z 866.934,A -85,B 0,C 180,E1 -20220.947,E2 -20220.947} C_VEL
LIN {X 0,Y 231.039,Z 877.038,A -85,B 0,C 180,E1 -20222.852,E2 -20222.852} C_VEL
LIN {X 0,Y 228.301,Z 886.304,A -85,B 0,C 180,E1 -20224.958,E2 -20224.958} C_VEL
LIN {X 0,Y 225.624,Z 895.599,A -85,B 0,C 180,E1 -20227.568,E2 -20227.568} C_VEL
LIN {X 0,Y 223.37,Z 903.343,A -85,B 0,C 180,E1 -20230.231,E2 -20230.231} C_VEL
LIN {X 0,Y 221.456,Z 910.736,A -85,B 0,C 180,E1 -20233.404,E2 -20233.404} C_VEL
LIN {X 0,Y 220.142,Z 915.906,A -85,B 0,C 180,E1 -20236.147,E2 -20236.147} C_VEL
LIN {X 0,Y 219.068,Z 921.255,A -85,B 0,C 180,E1 -20239.837,E2 -20239.837} C_VEL
LIN {X 0,Y 218.702,Z 924.244,A -85,B 0,C 180,E1 -20242.615,E2 -20242.615} C_VEL
LIN {X 0,Y 218.61,Z 926.339,A -85,B 0,C 180,E1 -20245.276,E2 -20245.276} C_VEL
LIN {X 0,Y 218.65,Z 927.821,A -85,B 0,C 180,E1 -20248.158,E2 -20248.158} C_VEL
LIN {X 0,Y 218.73,Z 928.32,A -85,B 0,C 180,E1 -20250,E2 -20250} C_VEL
LIN {X 0,Y 218.637,Z 928.47,A -85,B 0,C 180,E1 -20251.842,E2 -20251.842} C_VEL
LIN {X 0,Y 218.565,Z 927.758,A -85,B 0,C 180,E1 -20255.535,E2 -20255.535} C_VEL
LIN {X 0,Y 218.945,Z 925.701,A -85,B 0,C 180,E1 -20259.236,E2 -20259.236} C_VEL
LIN {X 0,Y 219.865,Z 922.258,A -85,B 0,C 180,E1 -20262.93,E2 -20262.93} C_VEL
LIN {X 0,Y 221.682,Z 917.339,A -85,B 0,C 180,E1 -20266.578,E2 -20266.578} C_VEL
LIN {X 0,Y 223.615,Z 912.253,A -85,B 0,C 180,E1 -20269.462,E2 -20269.462} C_VEL
LIN {X 0,Y 226.615,Z 904.671,A -85,B 0,C 180,E1 -20272.809,E2 -20272.809} C_VEL
LIN {X 0,Y 230.087,Z 895.979,A -85,B 0,C 180,E1 -20275.802,E2 -20275.802} C_VEL
LIN {X 0,Y 233.653,Z 886.915,A -85,B 0,C 180,E1 -20278.277,E2 -20278.277} C_VEL
LIN {X 0,Y 237.586,Z 876.116,A -85,B 0,C 180,E1 -20280.642,E2 -20280.642} C_VEL
LIN {X 0,Y 241.119,Z 864.846,A -85,B 0,C 180,E1 -20282.631,E2 -20282.631} C_VEL
LIN {X 0,Y 244.652,Z 852.602,A -85,B 0,C 180,E1 -20284.316,E2 -20284.316} C_VEL
LIN {X 0,Y 248.014,Z 838.874,A -85,B 0,C 180,E1 -20285.764,E2 -20285.764} C_VEL
LIN {X 0,Y 250.664,Z 825.506,A -85,B 0,C 180,E1 -20286.82,E2 -20286.82} C_VEL
LIN {X 0,Y 252.803,Z 810.914,A -85,B 0,C 180,E1 -20287.643,E2 -20287.643} C_VEL
LIN {X 0,Y 254.118,Z 796.061,A -85,B 0,C 180,E1 -20288.182,E2 -20288.182} C_VEL
LIN {X 0,Y 257.49,Z 729.344,A -85,B 0,C 180,E1 -20289.962,E2 -20289.962} C_VEL
LIN {X 0,Y 256.748,Z 724.906,A -85,B 0,C 180,E1 -20290.275,E2 -20290.275} C_VEL
LIN {X 0,Y 250.006,Z 709.323,A -85,B 0,C 180,E1 -20292.304,E2 -20292.304} C_VEL
LIN {X 0,Y 243.01,Z 695.482,A -85,B 0,C 180,E1 -20294.515,E2 -20294.515} C_VEL
LIN {X 0,Y 236.126,Z 683.408,A -85,B 0,C 180,E1 -20296.85,E2 -20296.85} C_VEL
LIN {X 0,Y 232.367,Z 677.405,A -85,B 0,C 180,E1 -20298.206,E2 -20298.206} C_VEL
LIN {X 0,Y 229.678,Z 673.201,A -85,B 0,C 180,E1 -20299.224,E2 -20299.224} C_VEL
LIN {X 0,Y 226.185,Z 667.835,A -85,B 0,C 180,E1 -20300.616,E2 -20300.616} C_VEL
LIN {X 0,Y 223.411,Z 663.967,A -85,B 0,C 180,E1 -20301.765,E2 -20301.765} C_VEL
LIN {X 0,Y 222.651,Z 662.306,A -85,B 0,C 180,E1 -20302.205,E2 -20302.205} C_VEL
LIN {X 0,Y 220.822,Z 657.098,A -85,B 0,C 180,E1 -20305.841,E2 -20305.841} C_VEL
LIN {X 0,Y 220.868,Z 657.062,A -85,B 0,C 180,E1 -20309.395,E2 -20309.395} C_VEL
LIN {X 0,Y 220.896,Z 657.082,A -85,B 0,C 180,E1 -20313.55,E2 -20313.55} C_VEL
LIN {X 0,Y 220.879,Z 657.083,A -85,B 0,C 180,E1 -20317.554,E2 -20317.554} C_VEL
LIN {X 0,Y 220.985,Z 657.073,A -85,B 0,C 180,E1 -20322.571,E2 -20322.571} C_VEL
LIN {X 0,Y 221.013,Z 657.07,A -85,B 0,C 180,E1 -20327.139,E2 -20327.139} C_VEL
LIN {X 0,Y 221.206,Z 657.041,A -85,B 0,C 180,E1 -20330.86,E2 -20330.86} C_VEL
LIN {X 0,Y 221.273,Z 657.045,A -85,B 0,C 180,E1 -20332.702,E2 -20332.702} C_VEL
LIN {X 0,Y 221.513,Z 657.019,A -85,B 0,C 180,E1 -20338.182,E2 -20338.182} C_VEL
LIN {X 0,Y 221.514,Z 657.008,A -85,B 0,C 180,E1 -20341.819,E2 -20341.819} C_VEL
LIN {X 0,Y 221.261,Z 657.045,A -85,B 0,C 180,E1 -20347.3,E2 -20347.3} C_VEL
LIN {X 0,Y 221.069,Z 657.06,A -85,B 0,C 180,E1 -20350.997,E2 -20350.997} C_VEL
LIN {X 0,Y 220.998,Z 657.069,A -85,B 0,C 180,E1 -20354.739,E2 -20354.739} C_VEL
LIN {X 0,Y 220.922,Z 657.082,A -85,B 0,C 180,E1 -20358.55,E2 -20358.55} C_VEL
LIN {X 0,Y 220.872,Z 657.09,A -85,B 0,C 180,E1 -20362.667,E2 -20362.667} C_VEL
LIN {X 0,Y 220.867,Z 657.076,A -85,B 0,C 180,E1 -20367.006,E2 -20367.006} C_VEL
LIN {X 0,Y 220.818,Z 657.103,A -85,B 0,C 180,E1 -20372.216,E2 -20372.216} C_VEL
LIN {X 0,Y 220.791,Z 657.109,A -85,B 0,C 180,E1 -20372.49,E2 -20372.49} C_VEL
LIN {X 0,Y 221.611,Z 659.615,A -85,B 0,C 180,E1 -20372.934,E2 -20372.934} C_VEL
LIN {X 0,Y 223.582,Z 661.87,A -85,B 0,C 180,E1 -20373.762,E2 -20373.762} C_VEL
LIN {X 0,Y 224.731,Z 662.779,A -85,B 0,C 180,E1 -20374.208,E2 -20374.208} C_VEL
LIN {X 0,Y 226.627,Z 665.913,A -85,B 0,C 180,E1 -20375.01,E2 -20375.01} C_VEL
LIN {X 0,Y 228.643,Z 668.104,A -85,B 0,C 180,E1 -20375.776,E2 -20375.776} C_VEL
LIN {X 0,Y 231.352,Z 671.743,A -85,B 0,C 180,E1 -20376.797,E2 -20376.797} C_VEL
LIN {X 0,Y 238.404,Z 681.82,A -85,B 0,C 180,E1 -20379.28,E2 -20379.28} C_VEL
LIN {X 0,Y 245.309,Z 692.272,A -85,B 0,C 180,E1 -20381.493,E2 -20381.493} C_VEL
LIN {X 0,Y 251.997,Z 703.705,A -85,B 0,C 180,E1 -20383.496,E2 -20383.496} C_VEL
LIN {X 0,Y 258.133,Z 716.713,A -85,B 0,C 180,E1 -20385.28,E2 -20385.28} C_VEL
LIN {X 0,Y 254.495,Z 786.415,A -85,B 0,C 180,E1 -20387.154,E2 -20387.154} C_VEL
LIN {X 0,Y 253.038,Z 800.845,A -85,B 0,C 180,E1 -20387.794,E2 -20387.794} C_VEL
LIN {X 0,Y 250.949,Z 814.656,A -85,B 0,C 180,E1 -20388.709,E2 -20388.709} C_VEL
LIN {X 0,Y 248.281,Z 827.56,A -85,B 0,C 180,E1 -20389.844,E2 -20389.844} C_VEL
LIN {X 0,Y 245.492,Z 839.417,A -85,B 0,C 180,E1 -20391.227,E2 -20391.227} C_VEL
LIN {X 0,Y 242.107,Z 851.308,A -85,B 0,C 180,E1 -20392.962,E2 -20392.962} C_VEL
LIN {X 0,Y 238.582,Z 862.146,A -85,B 0,C 180,E1 -20394.941,E2 -20394.941} C_VEL
LIN {X 0,Y 234.916,Z 872.836,A -85,B 0,C 180,E1 -20397.418,E2 -20397.418} C_VEL
LIN {X 0,Y 231.451,Z 881.627,A -85,B 0,C 180,E1 -20399.932,E2 -20399.932} C_VEL
LIN {X 0,Y 228.384,Z 888.913,A -85,B 0,C 180,E1 -20402.51,E2 -20402.51} C_VEL
LIN {X 0,Y 225.851,Z 894.953,A -85,B 0,C 180,E1 -20405.16,E2 -20405.16} C_VEL
LIN {X 0,Y 223.084,Z 901.352,A -85,B 0,C 180,E1 -20408.759,E2 -20408.759} C_VEL
LIN {X 0,Y 221.044,Z 906.213,A -85,B 0,C 180,E1 -20412.525,E2 -20412.525} C_VEL
LIN {X 0,Y 219.929,Z 908.628,A -85,B 0,C 180,E1 -20415.188,E2 -20415.188} C_VEL
LIN {X 0,Y 219.004,Z 910.804,A -85,B 0,C 180,E1 -20418.899,E2 -20418.899} C_VEL
LIN {X 0,Y 218.692,Z 911.637,A -85,B 0,C 180,E1 -20422.615,E2 -20422.615} C_VEL
LIN {X 0,Y 218.679,Z 911.486,A -85,B 0,C 180,E1 -20425.074,E2 -20425.074} C_VEL
LIN {X 0,Y 218.714,Z 910.434,A -85,B 0,C 180,E1 -20428.159,E2 -20428.159} C_VEL
LIN {X 0,Y 219.011,Z 907.993,A -85,B 0,C 180,E1 -20431.839,E2 -20431.839} C_VEL
LIN {X 0,Y 219.871,Z 904.154,A -85,B 0,C 180,E1 -20435.503,E2 -20435.503} C_VEL
LIN {X 0,Y 221.435,Z 898.756,A -85,B 0,C 180,E1 -20439.131,E2 -20439.131} C_VEL
LIN {X 0,Y 222.951,Z 893.643,A -85,B 0,C 180,E1 -20441.824,E2 -20441.824} C_VEL
LIN {X 0,Y 224.993,Z 886.296,A -85,B 0,C 180,E1 -20444.934,E2 -20444.934} C_VEL
LIN {X 0,Y 227.374,Z 878.611,A -85,B 0,C 180,E1 -20447.54,E2 -20447.54} C_VEL
LIN {X 0,Y 230.19,Z 869.357,A -85,B 0,C 180,E1 -20450.089,E2 -20450.089} C_VEL
LIN {X 0,Y 233.041,Z 859.123,A -85,B 0,C 180,E1 -20452.38,E2 -20452.38} C_VEL
LIN {X 0,Y 235.76,Z 847.859,A -85,B 0,C 180,E1 -20454.432,E2 -20454.432} C_VEL
LIN {X 0,Y 238.172,Z 836.957,A -85,B 0,C 180,E1 -20456.036,E2 -20456.036} C_VEL
LIN {X 0,Y 240.46,Z 825.278,A -85,B 0,C 180,E1 -20457.409,E2 -20457.409} C_VEL
LIN {X 0,Y 242.684,Z 811.295,A -85,B 0,C 180,E1 -20458.662,E2 -20458.662} C_VEL
LIN {X 0,Y 244.23,Z 797.302,A -85,B 0,C 180,E1 -20459.584,E2 -20459.584} C_VEL
LIN {X 0,Y 245.271,Z 784.014,A -85,B 0,C 180,E1 -20460.155,E2 -20460.155} C_VEL
LIN {X 0,Y 248.727,Z 708.379,A -85,B 0,C 180,E1 -20462.242,E2 -20462.242} C_VEL
LIN {X 0,Y 242.917,Z 694.586,A -85,B 0,C 180,E1 -20463.715,E2 -20463.715} C_VEL
LIN {X 0,Y 235.555,Z 681.192,A -85,B 0,C 180,E1 -20465.573,E2 -20465.573} C_VEL
LIN {X 0,Y 228.396,Z 669.472,A -85,B 0,C 180,E1 -20467.492,E2 -20467.492} C_VEL
LIN {X 0,Y 223.796,Z 662.484,A -85,B 0,C 180,E1 -20468.799,E2 -20468.799} C_VEL
LIN {X 0,Y 222.902,Z 661.303,A -85,B 0,C 180,E1 -20469.055,E2 -20469.055} C_VEL
LIN {X 0,Y 221.257,Z 658.875,A -85,B 0,C 180,E1 -20469.544,E2 -20469.544} C_VEL
LIN {X 0,Y 220.788,Z 657.087,A -85,B 0,C 180,E1 -20469.768,E2 -20469.768} C_VEL
LIN {X 0,Y 220.766,Z 657.105,A -85,B 0,C 180,E1 -20474.456,E2 -20474.456} C_VEL
LIN {X 0,Y 220.752,Z 657.109,A -85,B 0,C 180,E1 -20478.042,E2 -20478.042} C_VEL
LIN {X 0,Y 220.827,Z 657.063,A -85,B 0,C 180,E1 -20482.793,E2 -20482.793} C_VEL
LIN {X 0,Y 220.815,Z 657.105,A -85,B 0,C 180,E1 -20487.243,E2 -20487.243} C_VEL
LIN {X 0,Y 220.807,Z 657.098,A -85,B 0,C 180,E1 -20491.482,E2 -20491.482} C_VEL
LIN {X 0,Y 220.849,Z 657.08,A -85,B 0,C 180,E1 -20495.562,E2 -20495.562} C_VEL
LIN {X 0,Y 220.881,Z 657.095,A -85,B 0,C 180,E1 -20499.512,E2 -20499.512} C_VEL
LIN {X 0,Y 220.982,Z 657.062,A -85,B 0,C 180,E1 -20503.367,E2 -20503.367} C_VEL
LIN {X 0,Y 220.999,Z 657.076,A -85,B 0,C 180,E1 -20507.137,E2 -20507.137} C_VEL
LIN {X 0,Y 221.199,Z 657.038,A -85,B 0,C 180,E1 -20510.859,E2 -20510.859} C_VEL
LIN {X 0,Y 221.126,Z 657.062,A -85,B 0,C 180,E1 -20514.528,E2 -20514.528} C_VEL
LIN {X 0,Y 221.511,Z 657.019,A -85,B 0,C 180,E1 -20518.181,E2 -20518.181} C_VEL
LIN {X 0,Y 221.514,Z 657.008,A -85,B 0,C 180,E1 -20521.818,E2 -20521.818} C_VEL
LIN {X 0,Y 221.261,Z 657.045,A -85,B 0,C 180,E1 -20527.299,E2 -20527.299} C_VEL
LIN {X 0,Y 221.07,Z 657.061,A -85,B 0,C 180,E1 -20530.996,E2 -20530.996} C_VEL
LIN {X 0,Y 220.998,Z 657.072,A -85,B 0,C 180,E1 -20534.738,E2 -20534.738} C_VEL
LIN {X 0,Y 220.922,Z 657.084,A -85,B 0,C 180,E1 -20538.549,E2 -20538.549} C_VEL
LIN {X 0,Y 220.887,Z 657.089,A -85,B 0,C 180,E1 -20542.675,E2 -20542.675} C_VEL
LIN {X 0,Y 220.851,Z 657.09,A -85,B 0,C 180,E1 -20544.757,E2 -20544.757} C_VEL
LIN {X 0,Y 220.153,Z 657.182,A -85,B 0,C 180,E1 -20546.278,E2 -20546.278} C_VEL
LIN {X 0,Y 217.277,Z 657.543,A -85,B 0,C 180,E1 -20548.762,E2 -20548.762} C_VEL
LIN {X 0,Y 214.851,Z 657.842,A -85,B 0,C 180,E1 -20550.791,E2 -20550.791} C_VEL
LIN {X 0,Y 213.816,Z 657.977,A -85,B 0,C 180,E1 -20552.366,E2 -20552.366} C_VEL
LIN {X 0,Y 213.734,Z 657.977,A -85,B 0,C 180,E1 -20552.9,E2 -20552.9} C_VEL
LIN {X 0,Y 213.755,Z 657.981,A -85,B 0,C 180,E1 -20556.286,E2 -20556.286} C_VEL
LIN {X 0,Y 213.81,Z 658.084,A -85,B 0,C 180,E1 -20560.885,E2 -20560.885} C_VEL
LIN {X 0,Y 215.437,Z 663.551,A -85,B 0,C 180,E1 -20563.726,E2 -20563.726} C_VEL
LIN {X 0,Y 218.088,Z 668.083,A -85,B 0,C 180,E1 -20564.588,E2 -20564.588} C_VEL
LIN {X 0,Y 224.783,Z 680.15,A -85,B 0,C 180,E1 -20566.654,E2 -20566.654} C_VEL
LIN {X 0,Y 230.402,Z 691.077,A -85,B 0,C 180,E1 -20568.283,E2 -20568.283} C_VEL
LIN {X 0,Y 237.199,Z 706.714,A -85,B 0,C 180,E1 -20570.196,E2 -20570.196} C_VEL
LIN {X 0,Y 240.887,Z 716.523,A -85,B 0,C 180,E1 -20571.217,E2 -20571.217} C_VEL
LIN {X 0,Y 242.23,Z 728.468,A -85,B 0,C 180,E1 -20571.879,E2 -20571.879} C_VEL
LIN {X 0,Y 238.663,Z 802.637,A -85,B 0,C 180,E1 -20573.982,E2 -20573.982} C_VEL
LIN {X 0,Y 237.146,Z 817.336,A -85,B 0,C 180,E1 -20574.697,E2 -20574.697} C_VEL
LIN {X 0,Y 235.186,Z 830.795,A -85,B 0,C 180,E1 -20575.664,E2 -20575.664} C_VEL
LIN {X 0,Y 232.832,Z 843.053,A -85,B 0,C 180,E1 -20576.831,E2 -20576.831} C_VEL
LIN {X 0,Y 229.987,Z 855.955,A -85,B 0,C 180,E1 -20578.445,E2 -20578.445} C_VEL
LIN {X 0,Y 227.098,Z 867.689,A -85,B 0,C 180,E1 -20580.32,E2 -20580.32} C_VEL
LIN {X 0,Y 224.71,Z 876.461,A -85,B 0,C 180,E1 -20582.021,E2 -20582.021} C_VEL
LIN {X 0,Y 221.322,Z 887.42,A -85,B 0,C 180,E1 -20584.615,E2 -20584.615} C_VEL
LIN {X 0,Y 218.606,Z 896.484,A -85,B 0,C 180,E1 -20587.307,E2 -20587.307} C_VEL
LIN {X 0,Y 215.932,Z 905.153,A -85,B 0,C 180,E1 -20590.512,E2 -20590.512} C_VEL
LIN {X 0,Y 214.081,Z 912.154,A -85,B 0,C 180,E1 -20593.797,E2 -20593.797} C_VEL
LIN {X 0,Y 212.794,Z 916.981,A -85,B 0,C 180,E1 -20596.633,E2 -20596.633} C_VEL
LIN {X 0,Y 211.881,Z 921.98,A -85,B 0,C 180,E1 -20600.453,E2 -20600.453} C_VEL
LIN {X 0,Y 211.563,Z 925.46,A -85,B 0,C 180,E1 -20604.28,E2 -20604.28} C_VEL
LIN {X 0,Y 211.565,Z 927.518,A -85,B 0,C 180,E1 -20608.096,E2 -20608.096} C_VEL
LIN {X 0,Y 211.642,Z 928.031,A -85,B 0,C 180,E1 -20610,E2 -20610} C_VEL
LIN {X 0,Y 211.552,Z 928.195,A -85,B 0,C 180,E1 -20611.904,E2 -20611.904} C_VEL
LIN {X 0,Y 211.484,Z 927.511,A -85,B 0,C 180,E1 -20615.721,E2 -20615.721} C_VEL
LIN {X 0,Y 211.889,Z 925.482,A -85,B 0,C 180,E1 -20619.546,E2 -20619.546} C_VEL
LIN {X 0,Y 212.904,Z 922.065,A -85,B 0,C 180,E1 -20623.36,E2 -20623.36} C_VEL
LIN {X 0,Y 214.842,Z 917.175,A -85,B 0,C 180,E1 -20627.122,E2 -20627.122} C_VEL
LIN {X 0,Y 216.724,Z 912.536,A -85,B 0,C 180,E1 -20629.879,E2 -20629.879} C_VEL
LIN {X 0,Y 219.581,Z 905.69,A -85,B 0,C 180,E1 -20633.084,E2 -20633.084} C_VEL
LIN {X 0,Y 223.127,Z 897.272,A -85,B 0,C 180,E1 -20636.166,E2 -20636.166} C_VEL
LIN {X 0,Y 226.777,Z 888.521,A -85,B 0,C 180,E1 -20638.709,E2 -20638.709} C_VEL
LIN {X 0,Y 230.82,Z 877.94,A -85,B 0,C 180,E1 -20641.172,E2 -20641.172} C_VEL
LIN {X 0,Y 234.409,Z 867.284,A -85,B 0,C 180,E1 -20643.173,E2 -20643.173} C_VEL
LIN {X 0,Y 237.99,Z 855.677,A -85,B 0,C 180,E1 -20644.901,E2 -20644.901} C_VEL
LIN {X 0,Y 241.391,Z 842.926,A -85,B 0,C 180,E1 -20646.385,E2 -20646.385} C_VEL
LIN {X 0,Y 244.336,Z 829.709,A -85,B 0,C 180,E1 -20647.548,E2 -20647.548} C_VEL
LIN {X 0,Y 246.801,Z 815.376,A -85,B 0,C 180,E1 -20648.465,E2 -20648.465} C_VEL
LIN {X 0,Y 248.376,Z 801.137,A -85,B 0,C 180,E1 -20649.079,E2 -20649.079} C_VEL
LIN {X 0,Y 252.245,Z 730.852,A -85,B 0,C 180,E1 -20650.984,E2 -20650.984} C_VEL
LIN {X 0,Y 251.672,Z 727.755,A -85,B 0,C 180,E1 -20651.224,E2 -20651.224} C_VEL
LIN {X 0,Y 245.431,Z 713.166,A -85,B 0,C 180,E1 -20653.198,E2 -20653.198} C_VEL
LIN {X 0,Y 238.097,Z 698.481,A -85,B 0,C 180,E1 -20655.644,E2 -20655.644} C_VEL
LIN {X 0,Y 230.15,Z 684.557,A -85,B 0,C 180,E1 -20658.528,E2 -20658.528} C_VEL
LIN {X 0,Y 226.186,Z 678.429,A -85,B 0,C 180,E1 -20660.075,E2 -20660.075} C_VEL
LIN {X 0,Y 222.917,Z 673.316,A -85,B 0,C 180,E1 -20661.439,E2 -20661.439} C_VEL
LIN {X 0,Y 220.13,Z 669.232,A -85,B 0,C 180,E1 -20662.656,E2 -20662.656} C_VEL
LIN {X 0,Y 219.027,Z 667.599,A -85,B 0,C 180,E1 -20663.158,E2 -20663.158} C_VEL
LIN {X 0,Y 215.484,Z 662.748,A -85,B 0,C 180,E1 -20664.826,E2 -20664.826} C_VEL
LIN {X 0,Y 214.966,Z 661.766,A -85,B 0,C 180,E1 -20665.192,E2 -20665.192} C_VEL
LIN {X 0,Y 213.771,Z 657.944,A -85,B 0,C 180,E1 -20668.125,E2 -20668.125} C_VEL
LIN {X 0,Y 213.826,Z 657.968,A -85,B 0,C 180,E1 -20672.604,E2 -20672.604} C_VEL
LIN {X 0,Y 213.853,Z 657.96,A -85,B 0,C 180,E1 -20676.953,E2 -20676.953} C_VEL
LIN {X 0,Y 213.944,Z 657.951,A -85,B 0,C 180,E1 -20682.804,E2 -20682.804} C_VEL
LIN {X 0,Y 213.954,Z 657.946,A -85,B 0,C 180,E1 -20686.707,E2 -20686.707} C_VEL
LIN {X 0,Y 214.143,Z 657.921,A -85,B 0,C 180,E1 -20690.556,E2 -20690.556} C_VEL
LIN {X 0,Y 214.21,Z 657.922,A -85,B 0,C 180,E1 -20692.459,E2 -20692.459} C_VEL
LIN {X 0,Y 214.446,Z 657.899,A -85,B 0,C 180,E1 -20698.122,E2 -20698.122} C_VEL
LIN {X 0,Y 214.548,Z 657.872,A -85,B 0,C 180,E1 -20700.001,E2 -20700.001} C_VEL
LIN {X 0,Y 214.447,Z 657.888,A -85,B 0,C 180,E1 -20701.879,E2 -20701.879} C_VEL
LIN {X 0,Y 214.2,Z 657.928,A -85,B 0,C 180,E1 -20707.542,E2 -20707.542} C_VEL
LIN {X 0,Y 214.001,Z 657.943,A -85,B 0,C 180,E1 -20711.365,E2 -20711.365} C_VEL
LIN {X 0,Y 213.935,Z 657.948,A -85,B 0,C 180,E1 -20715.237,E2 -20715.237} C_VEL
LIN {X 0,Y 213.934,Z 657.961,A -85,B 0,C 180,E1 -20717.696,E2 -20717.696} C_VEL
LIN {X 0,Y 213.805,Z 657.967,A -85,B 0,C 180,E1 -20723.233,E2 -20723.233} C_VEL
LIN {X 0,Y 213.789,Z 657.95,A -85,B 0,C 180,E1 -20727.429,E2 -20727.429} C_VEL
LIN {X 0,Y 213.755,Z 658.003,A -85,B 0,C 180,E1 -20729.742,E2 -20729.742} C_VEL
LIN {X 0,Y 214.574,Z 660.467,A -85,B 0,C 180,E1 -20730.239,E2 -20730.239} C_VEL
LIN {X 0,Y 216.719,Z 662.888,A -85,B 0,C 180,E1 -20731.257,E2 -20731.257} C_VEL
LIN {X 0,Y 217.854,Z 663.746,A -85,B 0,C 180,E1 -20731.753,E2 -20731.753} C_VEL
LIN {X 0,Y 219.773,Z 666.884,A -85,B 0,C 180,E1 -20732.66,E2 -20732.66} C_VEL
LIN {X 0,Y 221.949,Z 669.162,A -85,B 0,C 180,E1 -20733.576,E2 -20733.576} C_VEL
LIN {X 0,Y 224.482,Z 672.678,A -85,B 0,C 180,E1 -20734.642,E2 -20734.642} C_VEL
LIN {X 0,Y 226.054,Z 674.728,A -85,B 0,C 180,E1 -20735.272,E2 -20735.272} C_VEL
LIN {X 0,Y 229.185,Z 679.073,A -85,B 0,C 180,E1 -20736.488,E2 -20736.488} C_VEL
LIN {X 0,Y 234.833,Z 687.104,A -85,B 0,C 180,E1 -20738.535,E2 -20738.535} C_VEL
LIN {X 0,Y 241.681,Z 697.726,A -85,B 0,C 180,E1 -20740.825,E2 -20740.825} C_VEL
LIN {X 0,Y 247.638,Z 708.035,A -85,B 0,C 180,E1 -20742.686,E2 -20742.686} C_VEL
LIN {X 0,Y 252.775,Z 718.983,A -85,B 0,C 180,E1 -20744.253,E2 -20744.253} C_VEL
LIN {X 0,Y 249.089,Z 787.359,A -85,B 0,C 180,E1 -20746.13,E2 -20746.13} C_VEL
LIN {X 0,Y 247.553,Z 801.473,A -85,B 0,C 180,E1 -20746.772,E2 -20746.772} C_VEL
LIN {X 0,Y 245.401,Z 815.192,A -85,B 0,C 180,E1 -20747.7,E2 -20747.7} C_VEL
LIN {X 0,Y 242.567,Z 828.33,A -85,B 0,C 180,E1 -20748.879,E2 -20748.879} C_VEL
LIN {X 0,Y 239.547,Z 840.571,A -85,B 0,C 180,E1 -20750.348,E2 -20750.348} C_VEL
LIN {X 0,Y 236.034,Z 852.304,A -85,B 0,C 180,E1 -20752.112,E2 -20752.112} C_VEL
LIN {X 0,Y 232.743,Z 862.039,A -85,B 0,C 180,E1 -20753.926,E2 -20753.926} C_VEL
LIN {X 0,Y 229.297,Z 871.666,A -85,B 0,C 180,E1 -20756.152,E2 -20756.152} C_VEL
LIN {X 0,Y 225.246,Z 881.637,A -85,B 0,C 180,E1 -20759.014,E2 -20759.014} C_VEL
LIN {X 0,Y 221.54,Z 890.087,A -85,B 0,C 180,E1 -20762.101,E2 -20762.101} C_VEL
LIN {X 0,Y 218.529,Z 896.857,A -85,B 0,C 180,E1 -20765.286,E2 -20765.286} C_VEL
LIN {X 0,Y 216.38,Z 901.489,A -85,B 0,C 180,E1 -20768.067,E2 -20768.067} C_VEL
LIN {X 0,Y 214.676,Z 905.215,A -85,B 0,C 180,E1 -20770.891,E2 -20770.891} C_VEL
LIN {X 0,Y 213.791,Z 907.205,A -85,B 0,C 180,E1 -20772.791,E2 -20772.791} C_VEL
LIN {X 0,Y 212.36,Z 910.109,A -85,B 0,C 180,E1 -20776.605,E2 -20776.605} C_VEL
LIN {X 0,Y 211.723,Z 911.638,A -85,B 0,C 180,E1 -20780.447,E2 -20780.447} C_VEL
LIN {X 0,Y 211.568,Z 911.843,A -85,B 0,C 180,E1 -20784.281,E2 -20784.281} C_VEL
LIN {X 0,Y 211.626,Z 910.746,A -85,B 0,C 180,E1 -20788.097,E2 -20788.097} C_VEL
LIN {X 0,Y 211.945,Z 908.335,A -85,B 0,C 180,E1 -20791.9,E2 -20791.9} C_VEL
LIN {X 0,Y 212.838,Z 904.537,A -85,B 0,C 180,E1 -20795.685,E2 -20795.685} C_VEL
LIN {X 0,Y 214.463,Z 899.184,A -85,B 0,C 180,E1 -20799.431,E2 -20799.431} C_VEL
LIN {X 0,Y 216.183,Z 893.618,A -85,B 0,C 180,E1 -20802.442,E2 -20802.442} C_VEL
LIN {X 0,Y 218.164,Z 886.799,A -85,B 0,C 180,E1 -20805.413,E2 -20805.413} C_VEL
LIN {X 0,Y 220.632,Z 879.149,A -85,B 0,C 180,E1 -20808.094,E2 -20808.094} C_VEL
LIN {X 0,Y 223.572,Z 869.957,A -85,B 0,C 180,E1 -20810.711,E2 -20810.711} C_VEL
LIN {X 0,Y 226.54,Z 859.801,A -85,B 0,C 180,E1 -20813.059,E2 -20813.059} C_VEL
LIN {X 0,Y 229.365,Z 848.628,A -85,B 0,C 180,E1 -20815.16,E2 -20815.16} C_VEL
LIN {X 0,Y 231.865,Z 837.827,A -85,B 0,C 180,E1 -20816.8,E2 -20816.8} C_VEL
LIN {X 0,Y 234.223,Z 826.268,A -85,B 0,C 180,E1 -20818.203,E2 -20818.203} C_VEL
LIN {X 0,Y 236.545,Z 812.567,A -85,B 0,C 180,E1 -20819.478,E2 -20819.478} C_VEL
LIN {X 0,Y 238.152,Z 798.981,A -85,B 0,C 180,E1 -20820.417,E2 -20820.417} C_VEL
LIN {X 0,Y 239.294,Z 785.12,A -85,B 0,C 180,E1 -20821.052,E2 -20821.052} C_VEL
LIN {X 0,Y 242.877,Z 710.277,A -85,B 0,C 180,E1 -20823.156,E2 -20823.156} C_VEL
LIN {X 0,Y 237.696,Z 698.068,A -85,B 0,C 180,E1 -20824.529,E2 -20824.529} C_VEL
LIN {X 0,Y 230.45,Z 684.705,A -85,B 0,C 180,E1 -20826.453,E2 -20826.453} C_VEL
LIN {X 0,Y 223.728,Z 673.855,A -85,B 0,C 180,E1 -20828.336,E2 -20828.336} C_VEL
LIN {X 0,Y 218.899,Z 666.534,A -85,B 0,C 180,E1 -20829.776,E2 -20829.776} C_VEL
LIN {X 0,Y 216.717,Z 663.038,A -85,B 0,C 180,E1 -20830.467,E2 -20830.467} C_VEL
LIN {X 0,Y 214.577,Z 660.618,A -85,B 0,C 180,E1 -20831.121,E2 -20831.121} C_VEL
LIN {X 0,Y 213.707,Z 657.98,A -85,B 0,C 180,E1 -20831.533,E2 -20831.533} C_VEL
LIN {X 0,Y 213.704,Z 657.986,A -85,B 0,C 180,E1 -20836.345,E2 -20836.345} C_VEL
LIN {X 0,Y 213.705,Z 657.99,A -85,B 0,C 180,E1 -20839.147,E2 -20839.147} C_VEL
LIN {X 0,Y 213.743,Z 657.948,A -85,B 0,C 180,E1 -20843.711,E2 -20843.711} C_VEL
LIN {X 0,Y 213.761,Z 657.975,A -85,B 0,C 180,E1 -20848.261,E2 -20848.261} C_VEL
LIN {X 0,Y 213.791,Z 657.979,A -85,B 0,C 180,E1 -20852.598,E2 -20852.598} C_VEL
LIN {X 0,Y 213.813,Z 657.96,A -85,B 0,C 180,E1 -20856.979,E2 -20856.979} C_VEL
LIN {X 0,Y 213.889,Z 657.942,A -85,B 0,C 180,E1 -20862.343,E2 -20862.343} C_VEL
LIN {X 0,Y 213.939,Z 657.959,A -85,B 0,C 180,E1 -20866.705,E2 -20866.705} C_VEL
LIN {X 0,Y 214.138,Z 657.914,A -85,B 0,C 180,E1 -20870.554,E2 -20870.554} C_VEL
LIN {X 0,Y 214.088,Z 657.939,A -85,B 0,C 180,E1 -20874.348,E2 -20874.348} C_VEL
LIN {X 0,Y 214.444,Z 657.899,A -85,B 0,C 180,E1 -20878.121,E2 -20878.121} C_VEL
LIN {X 0,Y 214.548,Z 657.876,A -85,B 0,C 180,E1 -20879.999,E2 -20879.999} C_VEL
LIN {X 0,Y 214.447,Z 657.889,A -85,B 0,C 180,E1 -20881.878,E2 -20881.878} C_VEL
LIN {X 0,Y 214.201,Z 657.925,A -85,B 0,C 180,E1 -20887.541,E2 -20887.541} C_VEL
LIN {X 0,Y 214.001,Z 657.943,A -85,B 0,C 180,E1 -20891.364,E2 -20891.364} C_VEL
LIN {X 0,Y 213.936,Z 657.95,A -85,B 0,C 180,E1 -20895.236,E2 -20895.236} C_VEL
LIN {X 0,Y 213.838,Z 657.963,A -85,B 0,C 180,E1 -20899.187,E2 -20899.187} C_VEL
LIN {X 0,Y 213.812,Z 657.967,A -85,B 0,C 180,E1 -20903.231,E2 -20903.231} C_VEL
LIN {X 0,Y 213.83,Z 657.965,A -85,B 0,C 180,E1 -20907.449,E2 -20907.449} C_VEL
LIN {X 0,Y 213.781,Z 657.977,A -85,B 0,C 180,E1 -20911.735,E2 -20911.735} C_VEL
LIN {X 0,Y 213.734,Z 657.977,A -85,B 0,C 180,E1 -20912.9,E2 -20912.9} C_VEL
LIN {X 0,Y 213.056,Z 658.066,A -85,B 0,C 180,E1 -20913.948,E2 -20913.948} C_VEL
LIN {X 0,Y 210.214,Z 658.426,A -85,B 0,C 180,E1 -20915.594,E2 -20915.594} C_VEL
LIN {X 0,Y 207.377,Z 658.777,A -85,B 0,C 180,E1 -20917.285,E2 -20917.285} C_VEL
LIN {X 0,Y 206.747,Z 658.855,A -85,B 0,C 180,E1 -20918.38,E2 -20918.38} C_VEL
LIN {X 0,Y 206.77,Z 658.99,A -85,B 0,C 180,E1 -20919.419,E2 -20919.419} C_VEL
LIN {X 0,Y 208.046,Z 663.194,A -85,B 0,C 180,E1 -20921.73,E2 -20921.73} C_VEL
LIN {X 0,Y 210.805,Z 667.724,A -85,B 0,C 180,E1 -20922.706,E2 -20922.706} C_VEL
LIN {X 0,Y 217.295,Z 678.978,A -85,B 0,C 180,E1 -20924.875,E2 -20924.875} C_VEL
LIN {X 0,Y 224.222,Z 692.149,A -85,B 0,C 180,E1 -20927.027,E2 -20927.027} C_VEL
LIN {X 0,Y 231.477,Z 708.695,A -85,B 0,C 180,E1 -20929.186,E2 -20929.186} C_VEL
LIN {X 0,Y 235.341,Z 719.053,A -85,B 0,C 180,E1 -20930.315,E2 -20930.315} C_VEL
LIN {X 0,Y 236.451,Z 729.385,A -85,B 0,C 180,E1 -20930.903,E2 -20930.903} C_VEL
LIN {X 0,Y 232.835,Z 802.062,A -85,B 0,C 180,E1 -20933.001,E2 -20933.001} C_VEL
LIN {X 0,Y 231.266,Z 816.876,A -85,B 0,C 180,E1 -20933.726,E2 -20933.726} C_VEL
LIN {X 0,Y 229.524,Z 828.674,A -85,B 0,C 180,E1 -20934.559,E2 -20934.559} C_VEL
LIN {X 0,Y 226.882,Z 842.226,A -85,B 0,C 180,E1 -20935.844,E2 -20935.844} C_VEL
LIN {X 0,Y 223.904,Z 855.233,A -85,B 0,C 180,E1 -20937.484,E2 -20937.484} C_VEL
LIN {X 0,Y 220.909,Z 867.048,A -85,B 0,C 180,E1 -20939.401,E2 -20939.401} C_VEL
LIN {X 0,Y 218.383,Z 875.878,A -85,B 0,C 180,E1 -20941.136,E2 -20941.136} C_VEL
LIN {X 0,Y 214.881,Z 886.892,A -85,B 0,C 180,E1 -20943.798,E2 -20943.798} C_VEL
LIN {X 0,Y 211.998,Z 895.997,A -85,B 0,C 180,E1 -20946.558,E2 -20946.558} C_VEL
LIN {X 0,Y 209.183,Z 904.702,A -85,B 0,C 180,E1 -20949.856,E2 -20949.856} C_VEL
LIN {X 0,Y 207.201,Z 911.737,A -85,B 0,C 180,E1 -20953.243,E2 -20953.243} C_VEL
LIN {X 0,Y 205.846,Z 916.595,A -85,B 0,C 180,E1 -20956.173,E2 -20956.173} C_VEL
LIN {X 0,Y 204.839,Z 921.623,A -85,B 0,C 180,E1 -20960.122,E2 -20960.122} C_VEL
LIN {X 0,Y 204.483,Z 925.13,A -85,B 0,C 180,E1 -20964.082,E2 -20964.082} C_VEL
LIN {X 0,Y 204.462,Z 927.213,A -85,B 0,C 180,E1 -20968.03,E2 -20968.03} C_VEL
LIN {X 0,Y 204.557,Z 927.74,A -85,B 0,C 180,E1 -20970,E2 -20970} C_VEL
LIN {X 0,Y 204.383,Z 927.757,A -85,B 0,C 180,E1 -20973.943,E2 -20973.943} C_VEL
LIN {X 0,Y 204.546,Z 926.432,A -85,B 0,C 180,E1 -20977.899,E2 -20977.899} C_VEL
LIN {X 0,Y 205.319,Z 923.745,A -85,B 0,C 180,E1 -20981.851,E2 -20981.851} C_VEL
LIN {X 0,Y 206.918,Z 919.634,A -85,B 0,C 180,E1 -20985.767,E2 -20985.767} C_VEL
LIN {X 0,Y 209.371,Z 913.984,A -85,B 0,C 180,E1 -20989.613,E2 -20989.613} C_VEL
LIN {X 0,Y 212.09,Z 907.635,A -85,B 0,C 180,E1 -20992.914,E2 -20992.914} C_VEL
LIN {X 0,Y 215.633,Z 899.766,A -85,B 0,C 180,E1 -20996.104,E2 -20996.104} C_VEL
LIN {X 0,Y 219.217,Z 891.567,A -85,B 0,C 180,E1 -20998.744,E2 -20998.744} C_VEL
LIN {X 0,Y 223.335,Z 881.712,A -85,B 0,C 180,E1 -21001.28,E2 -21001.28} C_VEL
LIN {X 0,Y 227.04,Z 871.543,A -85,B 0,C 180,E1 -21003.406,E2 -21003.406} C_VEL
LIN {X 0,Y 230.93,Z 859.968,A -85,B 0,C 180,E1 -21005.326,E2 -21005.326} C_VEL
LIN {X 0,Y 234.431,Z 848.306,A -85,B 0,C 180,E1 -21006.84,E2 -21006.84} C_VEL
LIN {X 0,Y 237.846,Z 834.608,A -85,B 0,C 180,E1 -21008.219,E2 -21008.219} C_VEL
LIN {X 0,Y 240.539,Z 820.63,A -85,B 0,C 180,E1 -21009.253,E2 -21009.253} C_VEL
LIN {X 0,Y 242.543,Z 806.73,A -85,B 0,C 180,E1 -21009.952,E2 -21009.952} C_VEL
LIN {X 0,Y 243.806,Z 789.945,A -85,B 0,C 180,E1 -21010.5,E2 -21010.5} C_VEL
LIN {X 0,Y 247.042,Z 732.089,A -85,B 0,C 180,E1 -21012.068,E2 -21012.068} C_VEL
LIN {X 0,Y 244.203,Z 724.679,A -85,B 0,C 180,E1 -21013.017,E2 -21013.017} C_VEL
LIN {X 0,Y 239.232,Z 713.467,A -85,B 0,C 180,E1 -21014.7,E2 -21014.7} C_VEL
LIN {X 0,Y 233.36,Z 701.831,A -85,B 0,C 180,E1 -21016.783,E2 -21016.783} C_VEL
LIN {X 0,Y 227.683,Z 691.696,A -85,B 0,C 180,E1 -21018.937,E2 -21018.937} C_VEL
LIN {X 0,Y 223.134,Z 684.19,A -85,B 0,C 180,E1 -21020.792,E2 -21020.792} C_VEL
LIN {X 0,Y 219.613,Z 678.713,A -85,B 0,C 180,E1 -21022.322,E2 -21022.322} C_VEL
LIN {X 0,Y 215.907,Z 673.148,A -85,B 0,C 180,E1 -21024.042,E2 -21024.042} C_VEL
LIN {X 0,Y 211.57,Z 667.067,A -85,B 0,C 180,E1 -21026.214,E2 -21026.214} C_VEL
LIN {X 0,Y 208.418,Z 662.89,A -85,B 0,C 180,E1 -21027.927,E2 -21027.927} C_VEL
LIN {X 0,Y 207.546,Z 661.318,A -85,B 0,C 180,E1 -21028.509,E2 -21028.509} C_VEL
LIN {X 0,Y 206.739,Z 658.836,A -85,B 0,C 180,E1 -21030.747,E2 -21030.747} C_VEL
LIN {X 0,Y 206.764,Z 658.852,A -85,B 0,C 180,E1 -21035.928,E2 -21035.928} C_VEL
LIN {X 0,Y 206.785,Z 658.85,A -85,B 0,C 180,E1 -21040.132,E2 -21040.132} C_VEL
LIN {X 0,Y 206.869,Z 658.842,A -85,B 0,C 180,E1 -21044.23,E2 -21044.23} C_VEL
LIN {X 0,Y 207.061,Z 658.807,A -85,B 0,C 180,E1 -21049.836,E2 -21049.836} C_VEL
LIN {X 0,Y 207.15,Z 658.798,A -85,B 0,C 180,E1 -21052.201,E2 -21052.201} C_VEL
LIN {X 0,Y 207.383,Z 658.778,A -85,B 0,C 180,E1 -21058.058,E2 -21058.058} C_VEL
LIN {X 0,Y 207.513,Z 658.748,A -85,B 0,C 180,E1 -21060.001,E2 -21060.001} C_VEL
LIN {X 0,Y 207.383,Z 658.768,A -85,B 0,C 180,E1 -21061.943,E2 -21061.943} C_VEL
LIN {X 0,Y 207.143,Z 658.808,A -85,B 0,C 180,E1 -21067.8,E2 -21067.8} C_VEL
LIN {X 0,Y 206.927,Z 658.827,A -85,B 0,C 180,E1 -21071.759,E2 -21071.759} C_VEL
LIN {X 0,Y 206.873,Z 658.829,A -85,B 0,C 180,E1 -21075.771,E2 -21075.771} C_VEL
LIN {X 0,Y 206.766,Z 658.842,A -85,B 0,C 180,E1 -21079.872,E2 -21079.872} C_VEL
LIN {X 0,Y 206.741,Z 658.847,A -85,B 0,C 180,E1 -21084.076,E2 -21084.076} C_VEL
LIN {X 0,Y 206.726,Z 658.89,A -85,B 0,C 180,E1 -21086.547,E2 -21086.547} C_VEL
LIN {X 0,Y 207.474,Z 661.203,A -85,B 0,C 180,E1 -21087.079,E2 -21087.079} C_VEL
LIN {X 0,Y 209.407,Z 663.569,A -85,B 0,C 180,E1 -21088.162,E2 -21088.162} C_VEL
LIN {X 0,Y 211.081,Z 664.8,A -85,B 0,C 180,E1 -21089.004,E2 -21089.004} C_VEL
LIN {X 0,Y 213.025,Z 667.963,A -85,B 0,C 180,E1 -21090.047,E2 -21090.047} C_VEL
LIN {X 0,Y 215.178,Z 670.078,A -85,B 0,C 180,E1 -21091.065,E2 -21091.065} C_VEL
LIN {X 0,Y 217.646,Z 673.548,A -85,B 0,C 180,E1 -21092.234,E2 -21092.234} C_VEL
LIN {X 0,Y 219.114,Z 675.248,A -85,B 0,C 180,E1 -21092.881,E2 -21092.881} C_VEL
LIN {X 0,Y 223.369,Z 681.06,A -85,B 0,C 180,E1 -21094.702,E2 -21094.702} C_VEL
LIN {X 0,Y 226.505,Z 685.487,A -85,B 0,C 180,E1 -21095.962,E2 -21095.962} C_VEL
LIN {X 0,Y 231.496,Z 692.734,A -85,B 0,C 180,E1 -21097.839,E2 -21097.839} C_VEL
LIN {X 0,Y 237.681,Z 702.495,A -85,B 0,C 180,E1 -21100,E2 -21100} C_VEL
LIN {X 0,Y 243.568,Z 712.905,A -85,B 0,C 180,E1 -21101.926,E2 -21101.926} C_VEL
LIN {X 0,Y 247.472,Z 721.273,A -85,B 0,C 180,E1 -21103.177,E2 -21103.177} C_VEL
LIN {X 0,Y 243.828,Z 787.326,A -85,B 0,C 180,E1 -21105.025,E2 -21105.025} C_VEL
LIN {X 0,Y 242.25,Z 801.505,A -85,B 0,C 180,E1 -21105.67,E2 -21105.67} C_VEL
LIN {X 0,Y 239.938,Z 815.732,A -85,B 0,C 180,E1 -21106.646,E2 -21106.646} C_VEL
LIN {X 0,Y 236.946,Z 829.043,A -85,B 0,C 180,E1 -21107.862,E2 -21107.862} C_VEL
LIN {X 0,Y 233.661,Z 841.729,A -85,B 0,C 180,E1 -21109.426,E2 -21109.426} C_VEL
LIN {X 0,Y 230.014,Z 853.305,A -85,B 0,C 180,E1 -21111.217,E2 -21111.217} C_VEL
LIN {X 0,Y 226.256,Z 863.897,A -85,B 0,C 180,E1 -21113.277,E2 -21113.277} C_VEL
LIN {X 0,Y 222.912,Z 872.753,A -85,B 0,C 180,E1 -21115.424,E2 -21115.424} C_VEL
LIN {X 0,Y 219.101,Z 881.65,A -85,B 0,C 180,E1 -21118.044,E2 -21118.044} C_VEL
LIN {X 0,Y 215.202,Z 890.144,A -85,B 0,C 180,E1 -21121.204,E2 -21121.204} C_VEL
LIN {X 0,Y 212.004,Z 896.956,A -85,B 0,C 180,E1 -21124.472,E2 -21124.472} C_VEL
LIN {X 0,Y 209.703,Z 901.626,A -85,B 0,C 180,E1 -21127.331,E2 -21127.331} C_VEL
LIN {X 0,Y 207.868,Z 905.387,A -85,B 0,C 180,E1 -21130.239,E2 -21130.239} C_VEL
LIN {X 0,Y 206.947,Z 907.394,A -85,B 0,C 180,E1 -21132.203,E2 -21132.203} C_VEL
LIN {X 0,Y 205.4,Z 910.33,A -85,B 0,C 180,E1 -21136.142,E2 -21136.142} C_VEL
LIN {X 0,Y 204.67,Z 911.889,A -85,B 0,C 180,E1 -21140.114,E2 -21140.114} C_VEL
LIN {X 0,Y 204.485,Z 912.124,A -85,B 0,C 180,E1 -21144.082,E2 -21144.082} C_VEL
LIN {X 0,Y 204.541,Z 911.057,A -85,B 0,C 180,E1 -21148.031,E2 -21148.031} C_VEL
LIN {X 0,Y 204.882,Z 908.677,A -85,B 0,C 180,E1 -21151.966,E2 -21151.966} C_VEL
LIN {X 0,Y 205.808,Z 904.915,A -85,B 0,C 180,E1 -21155.88,E2 -21155.88} C_VEL
LIN {X 0,Y 207.499,Z 899.611,A -85,B 0,C 180,E1 -21159.75,E2 -21159.75} C_VEL
LIN {X 0,Y 209.422,Z 893.676,A -85,B 0,C 180,E1 -21163.052,E2 -21163.052} C_VEL
LIN {X 0,Y 211.714,Z 886.1,A -85,B 0,C 180,E1 -21166.39,E2 -21166.39} C_VEL
LIN {X 0,Y 214.42,Z 878.269,A -85,B 0,C 180,E1 -21169.134,E2 -21169.134} C_VEL
LIN {X 0,Y 217.521,Z 868.825,A -85,B 0,C 180,E1 -21171.812,E2 -21171.812} C_VEL
LIN {X 0,Y 220.597,Z 858.377,A -85,B 0,C 180,E1 -21174.217,E2 -21174.217} C_VEL
LIN {X 0,Y 223.568,Z 846.845,A -85,B 0,C 180,E1 -21176.361,E2 -21176.361} C_VEL
LIN {X 0,Y 226.614,Z 834.013,A -85,B 0,C 180,E1 -21178.226,E2 -21178.226} C_VEL
LIN {X 0,Y 229.362,Z 820.445,A -85,B 0,C 180,E1 -21179.737,E2 -21179.737} C_VEL
LIN {X 0,Y 231.329,Z 807.385,A -85,B 0,C 180,E1 -21180.843,E2 -21180.843} C_VEL
LIN {X 0,Y 232.849,Z 793.245,A -85,B 0,C 180,E1 -21181.693,E2 -21181.693} C_VEL
LIN {X 0,Y 233.821,Z 778.36,A -85,B 0,C 180,E1 -21182.244,E2 -21182.244} C_VEL
LIN {X 0,Y 237.117,Z 712.293,A -85,B 0,C 180,E1 -21184.105,E2 -21184.105} C_VEL
LIN {X 0,Y 232.547,Z 701.642,A -85,B 0,C 180,E1 -21185.372,E2 -21185.372} C_VEL
LIN {X 0,Y 225.692,Z 688.909,A -85,B 0,C 180,E1 -21187.281,E2 -21187.281} C_VEL
LIN {X 0,Y 219.309,Z 678.445,A -85,B 0,C 180,E1 -21189.159,E2 -21189.159} C_VEL
LIN {X 0,Y 214.466,Z 671.084,A -85,B 0,C 180,E1 -21190.673,E2 -21190.673} C_VEL
LIN {X 0,Y 212.118,Z 667.687,A -85,B 0,C 180,E1 -21191.438,E2 -21191.438} C_VEL
LIN {X 0,Y 209.892,Z 664.302,A -85,B 0,C 180,E1 -21192.197,E2 -21192.197} C_VEL
LIN {X 0,Y 207.379,Z 661.214,A -85,B 0,C 180,E1 -21193.05,E2 -21193.05} C_VEL
LIN {X 0,Y 206.658,Z 658.863,A -85,B 0,C 180,E1 -21193.422,E2 -21193.422} C_VEL
LIN {X 0,Y 206.634,Z 658.87,A -85,B 0,C 180,E1 -21198.44,E2 -21198.44} C_VEL
LIN {X 0,Y 206.666,Z 658.827,A -85,B 0,C 180,E1 -21202.256,E2 -21202.256} C_VEL
LIN {X 0,Y 206.702,Z 658.835,A -85,B 0,C 180,E1 -21204.688,E2 -21204.688} C_VEL
LIN {X 0,Y 206.698,Z 658.846,A -85,B 0,C 180,E1 -21209.334,E2 -21209.334} C_VEL
LIN {X 0,Y 206.708,Z 658.857,A -85,B 0,C 180,E1 -21213.768,E2 -21213.768} C_VEL
LIN {X 0,Y 206.737,Z 658.852,A -85,B 0,C 180,E1 -21218.04,E2 -21218.04} C_VEL
LIN {X 0,Y 206.829,Z 658.822,A -85,B 0,C 180,E1 -21222.192,E2 -21222.192} C_VEL
LIN {X 0,Y 206.88,Z 658.839,A -85,B 0,C 180,E1 -21226.243,E2 -21226.243} C_VEL
LIN {X 0,Y 207.082,Z 658.791,A -85,B 0,C 180,E1 -21230.23,E2 -21230.23} C_VEL
LIN {X 0,Y 207.05,Z 658.816,A -85,B 0,C 180,E1 -21234.155,E2 -21234.155} C_VEL
LIN {X 0,Y 207.38,Z 658.779,A -85,B 0,C 180,E1 -21238.057,E2 -21238.057} C_VEL
LIN {X 0,Y 207.514,Z 658.753,A -85,B 0,C 180,E1 -21239.999,E2 -21239.999} C_VEL
LIN {X 0,Y 207.383,Z 658.769,A -85,B 0,C 180,E1 -21241.942,E2 -21241.942} C_VEL
LIN {X 0,Y 207.143,Z 658.806,A -85,B 0,C 180,E1 -21247.799,E2 -21247.799} C_VEL
LIN {X 0,Y 206.927,Z 658.826,A -85,B 0,C 180,E1 -21251.758,E2 -21251.758} C_VEL
LIN {X 0,Y 206.869,Z 658.83,A -85,B 0,C 180,E1 -21255.77,E2 -21255.77} C_VEL
LIN {X 0,Y 206.765,Z 658.843,A -85,B 0,C 180,E1 -21259.87,E2 -21259.87} C_VEL
LIN {X 0,Y 206.749,Z 658.846,A -85,B 0,C 180,E1 -21264.073,E2 -21264.073} C_VEL
LIN {X 0,Y 206.745,Z 658.851,A -85,B 0,C 180,E1 -21268.418,E2 -21268.418} C_VEL
LIN {X 0,Y 206.71,Z 658.861,A -85,B 0,C 180,E1 -21272.955,E2 -21272.955} C_VEL
LIN {X 0,Y 206.725,Z 658.858,A -85,B 0,C 180,E1 -21277.73,E2 -21277.73} C_VEL
LIN {X 0,Y 206.747,Z 658.855,A -85,B 0,C 180,E1 -21278.38,E2 -21278.38} C_VEL
LIN {X 0,Y 206.843,Z 659.548,A -85,B 0,C 180,E1 -21279.261,E2 -21279.261} C_VEL
LIN {X 0,Y 207.083,Z 661.853,A -85,B 0,C 180,E1 -21280.245,E2 -21280.245} C_VEL
LIN {X 0,Y 207.617,Z 666.365,A -85,B 0,C 180,E1 -21281.301,E2 -21281.301} C_VEL
LIN {X 0,Y 209.425,Z 675.698,A -85,B 0,C 180,E1 -21282.669,E2 -21282.669} C_VEL
LIN {X 0,Y 211.501,Z 681.011,A -85,B 0,C 180,E1 -21283.51,E2 -21283.51} C_VEL
LIN {X 0,Y 212.45,Z 682.555,A -85,B 0,C 180,E1 -21283.827,E2 -21283.827} C_VEL
LIN {X 0,Y 219.84,Z 696.959,A -85,B 0,C 180,E1 -21286.252,E2 -21286.252} C_VEL
LIN {X 0,Y 226.675,Z 712.898,A -85,B 0,C 180,E1 -21288.389,E2 -21288.389} C_VEL
LIN {X 0,Y 229.896,Z 721.723,A -85,B 0,C 180,E1 -21289.383,E2 -21289.383} C_VEL
LIN {X 0,Y 230.72,Z 731.111,A -85,B 0,C 180,E1 -21289.905,E2 -21289.905} C_VEL
LIN {X 0,Y 226.967,Z 802.66,A -85,B 0,C 180,E1 -21292.017,E2 -21292.017} C_VEL
LIN {X 0,Y 225.342,Z 817.17,A -85,B 0,C 180,E1 -21292.753,E2 -21292.753} C_VEL
LIN {X 0,Y 223.374,Z 829.967,A -85,B 0,C 180,E1 -21293.708,E2 -21293.708} C_VEL
LIN {X 0,Y 220.602,Z 843.169,A -85,B 0,C 180,E1 -21295.009,E2 -21295.009} C_VEL
LIN {X 0,Y 217.538,Z 855.944,A -85,B 0,C 180,E1 -21296.686,E2 -21296.686} C_VEL
LIN {X 0,Y 214.445,Z 867.587,A -85,B 0,C 180,E1 -21298.649,E2 -21298.649} C_VEL
LIN {X 0,Y 212.083,Z 875.289,A -85,B 0,C 180,E1 -21300.193,E2 -21300.193} C_VEL
LIN {X 0,Y 208.471,Z 886.359,A -85,B 0,C 180,E1 -21302.927,E2 -21302.927} C_VEL
LIN {X 0,Y 205.464,Z 895.51,A -85,B 0,C 180,E1 -21305.766,E2 -21305.766} C_VEL
LIN {X 0,Y 202.478,Z 904.253,A -85,B 0,C 180,E1 -21309.159,E2 -21309.159} C_VEL
LIN {X 0,Y 200.345,Z 911.32,A -85,B 0,C 180,E1 -21312.652,E2 -21312.652} C_VEL
LIN {X 0,Y 198.919,Z 916.21,A -85,B 0,C 180,E1 -21315.681,E2 -21315.681} C_VEL
LIN {X 0,Y 197.789,Z 921.264,A -85,B 0,C 180,E1 -21319.766,E2 -21319.766} C_VEL
LIN {X 0,Y 197.385,Z 924.799,A -85,B 0,C 180,E1 -21323.868,E2 -21323.868} C_VEL
LIN {X 0,Y 197.362,Z 926.909,A -85,B 0,C 180,E1 -21327.959,E2 -21327.959} C_VEL
LIN {X 0,Y 197.473,Z 927.448,A -85,B 0,C 180,E1 -21330,E2 -21330} C_VEL
LIN {X 0,Y 197.284,Z 927.49,A -85,B 0,C 180,E1 -21334.085,E2 -21334.085} C_VEL
LIN {X 0,Y 197.482,Z 926.194,A -85,B 0,C 180,E1 -21338.184,E2 -21338.184} C_VEL
LIN {X 0,Y 198.327,Z 923.539,A -85,B 0,C 180,E1 -21342.276,E2 -21342.276} C_VEL
LIN {X 0,Y 200.057,Z 919.456,A -85,B 0,C 180,E1 -21346.322,E2 -21346.322} C_VEL
LIN {X 0,Y 202.602,Z 913.834,A -85,B 0,C 180,E1 -21350.297,E2 -21350.297} C_VEL
LIN {X 0,Y 205.517,Z 907.519,A -85,B 0,C 180,E1 -21353.691,E2 -21353.691} C_VEL
LIN {X 0,Y 209.26,Z 899.686,A -85,B 0,C 180,E1 -21356.962,E2 -21356.962} C_VEL
LIN {X 0,Y 212.996,Z 891.527,A -85,B 0,C 180,E1 -21359.666,E2 -21359.666} C_VEL
LIN {X 0,Y 217.27,Z 881.719,A -85,B 0,C 180,E1 -21362.257,E2 -21362.257} C_VEL
LIN {X 0,Y 221.421,Z 870.855,A -85,B 0,C 180,E1 -21364.564,E2 -21364.564} C_VEL
LIN {X 0,Y 225.606,Z 858.811,A -85,B 0,C 180,E1 -21366.568,E2 -21366.568} C_VEL
LIN {X 0,Y 229.261,Z 846.951,A -85,B 0,C 180,E1 -21368.092,E2 -21368.092} C_VEL
LIN {X 0,Y 232.546,Z 833.951,A -85,B 0,C 180,E1 -21369.395,E2 -21369.395} C_VEL
LIN {X 0,Y 235.356,Z 819.796,A -85,B 0,C 180,E1 -21370.432,E2 -21370.432} C_VEL
LIN {X 0,Y 237.406,Z 805.456,A -85,B 0,C 180,E1 -21371.15,E2 -21371.15} C_VEL
LIN {X 0,Y 238.804,Z 786.973,A -85,B 0,C 180,E1 -21371.73,E2 -21371.73} C_VEL
LIN {X 0,Y 241.879,Z 733.963,A -85,B 0,C 180,E1 -21373.186,E2 -21373.186} C_VEL
LIN {X 0,Y 236.668,Z 721.355,A -85,B 0,C 180,E1 -21375.017,E2 -21375.017} C_VEL
LIN {X 0,Y 230.345,Z 708.134,A -85,B 0,C 180,E1 -21377.35,E2 -21377.35} C_VEL
LIN {X 0,Y 223.293,Z 695.172,A -85,B 0,C 180,E1 -21380.169,E2 -21380.169} C_VEL
LIN {X 0,Y 216.847,Z 684.669,A -85,B 0,C 180,E1 -21383.015,E2 -21383.015} C_VEL
LIN {X 0,Y 213.755,Z 679.834,A -85,B 0,C 180,E1 -21384.508,E2 -21384.508} C_VEL
LIN {X 0,Y 208.897,Z 672.971,A -85,B 0,C 180,E1 -21387.031,E2 -21387.031} C_VEL
LIN {X 0,Y 205.682,Z 668.463,A -85,B 0,C 180,E1 -21388.88,E2 -21388.88} C_VEL
LIN {X 0,Y 204.948,Z 667.367,A -85,B 0,C 180,E1 -21389.331,E2 -21389.331} C_VEL
LIN {X 0,Y 200.502,Z 662.204,A -85,B 0,C 180,E1 -21392.173,E2 -21392.173} C_VEL
LIN {X 0,Y 199.866,Z 660.608,A -85,B 0,C 180,E1 -21392.799,E2 -21392.799} C_VEL
LIN {X 0,Y 199.687,Z 659.723,A -85,B 0,C 180,E1 -21393.619,E2 -21393.619} C_VEL
LIN {X 0,Y 199.739,Z 659.716,A -85,B 0,C 180,E1 -21397.23,E2 -21397.23} C_VEL
LIN {X 0,Y 199.797,Z 659.709,A -85,B 0,C 180,E1 -21401.758,E2 -21401.758} C_VEL
LIN {X 0,Y 199.837,Z 659.704,A -85,B 0,C 180,E1 -21405.749,E2 -21405.749} C_VEL
LIN {X 0,Y 200.023,Z 659.683,A -85,B 0,C 180,E1 -21409.882,E2 -21409.882} C_VEL
LIN {X 0,Y 200.028,Z 659.69,A -85,B 0,C 180,E1 -21413.95,E2 -21413.95} C_VEL
LIN {X 0,Y 200.322,Z 659.657,A -85,B 0,C 180,E1 -21417.99,E2 -21417.99} C_VEL
LIN {X 0,Y 200.478,Z 659.623,A -85,B 0,C 180,E1 -21420.001,E2 -21420.001} C_VEL
LIN {X 0,Y 200.03,Z 659.686,A -85,B 0,C 180,E1 -21424.03,E2 -21424.03} C_VEL
LIN {X 0,Y 200.091,Z 659.687,A -85,B 0,C 180,E1 -21428.077,E2 -21428.077} C_VEL
LIN {X 0,Y 199.876,Z 659.709,A -85,B 0,C 180,E1 -21432.18,E2 -21432.18} C_VEL
LIN {X 0,Y 199.809,Z 659.713,A -85,B 0,C 180,E1 -21436.344,E2 -21436.344} C_VEL
LIN {X 0,Y 199.684,Z 659.729,A -85,B 0,C 180,E1 -21440.608,E2 -21440.608} C_VEL
LIN {X 0,Y 199.685,Z 659.739,A -85,B 0,C 180,E1 -21442.71,E2 -21442.71} C_VEL
LIN {X 0,Y 200.466,Z 662.132,A -85,B 0,C 180,E1 -21443.378,E2 -21443.378} C_VEL
LIN {X 0,Y 202.335,Z 664.444,A -85,B 0,C 180,E1 -21444.634,E2 -21444.634} C_VEL
LIN {X 0,Y 204.321,Z 665.784,A -85,B 0,C 180,E1 -21445.807,E2 -21445.807} C_VEL
LIN {X 0,Y 206.133,Z 668.843,A -85,B 0,C 180,E1 -21446.95,E2 -21446.95} C_VEL
LIN {X 0,Y 208.588,Z 671.125,A -85,B 0,C 180,E1 -21448.283,E2 -21448.283} C_VEL
LIN {X 0,Y 211.114,Z 674.724,A -85,B 0,C 180,E1 -21449.649,E2 -21449.649} C_VEL
LIN {X 0,Y 212.778,Z 676.598,A -85,B 0,C 180,E1 -21450.473,E2 -21450.473} C_VEL
LIN {X 0,Y 215.693,Z 680.349,A -85,B 0,C 180,E1 -21451.872,E2 -21451.872} C_VEL
LIN {X 0,Y 222.258,Z 689.427,A -85,B 0,C 180,E1 -21454.763,E2 -21454.763} C_VEL
LIN {X 0,Y 228.611,Z 699,A -85,B 0,C 180,E1 -21457.281,E2 -21457.281} C_VEL
LIN {X 0,Y 234.887,Z 709.22,A -85,B 0,C 180,E1 -21459.551,E2 -21459.551} C_VEL
LIN {X 0,Y 239.607,Z 717.875,A -85,B 0,C 180,E1 -21461.161,E2 -21461.161} C_VEL
LIN {X 0,Y 242.275,Z 723.678,A -85,B 0,C 180,E1 -21462.061,E2 -21462.061} C_VEL
LIN {X 0,Y 241.816,Z 733.897,A -85,B 0,C 180,E1 -21462.374,E2 -21462.374} C_VEL
LIN {X 0,Y 238.53,Z 788.68,A -85,B 0,C 180,E1 -21463.922,E2 -21463.922} C_VEL
LIN {X 0,Y 236.861,Z 802.738,A -85,B 0,C 180,E1 -21464.593,E2 -21464.593} C_VEL
LIN {X 0,Y 234.561,Z 816.272,A -85,B 0,C 180,E1 -21465.543,E2 -21465.543} C_VEL
LIN {X 0,Y 231.423,Z 829.699,A -85,B 0,C 180,E1 -21466.791,E2 -21466.791} C_VEL
LIN {X 0,Y 227.846,Z 842.888,A -85,B 0,C 180,E1 -21468.458,E2 -21468.458} C_VEL
LIN {X 0,Y 224.066,Z 854.305,A -85,B 0,C 180,E1 -21470.277,E2 -21470.277} C_VEL
LIN {X 0,Y 219.795,Z 865.747,A -85,B 0,C 180,E1 -21472.589,E2 -21472.589} C_VEL
LIN {X 0,Y 215.682,Z 875.912,A -85,B 0,C 180,E1 -21475.233,E2 -21475.233} C_VEL
LIN {X 0,Y 211.794,Z 884.316,A -85,B 0,C 180,E1 -21477.932,E2 -21477.932} C_VEL
LIN {X 0,Y 207.876,Z 892.315,A -85,B 0,C 180,E1 -21481.199,E2 -21481.199} C_VEL
LIN {X 0,Y 204.657,Z 898.728,A -85,B 0,C 180,E1 -21484.58,E2 -21484.58} C_VEL
LIN {X 0,Y 201.709,Z 904.387,A -85,B 0,C 180,E1 -21488.541,E2 -21488.541} C_VEL
LIN {X 0,Y 200.107,Z 907.583,A -85,B 0,C 180,E1 -21491.573,E2 -21491.573} C_VEL
LIN {X 0,Y 198.457,Z 910.55,A -85,B 0,C 180,E1 -21495.647,E2 -21495.647} C_VEL
LIN {X 0,Y 197.617,Z 912.141,A -85,B 0,C 180,E1 -21499.757,E2 -21499.757} C_VEL
LIN {X 0,Y 197.385,Z 912.406,A -85,B 0,C 180,E1 -21503.868,E2 -21503.868} C_VEL
LIN {X 0,Y 197.438,Z 911.369,A -85,B 0,C 180,E1 -21507.96,E2 -21507.96} C_VEL
LIN {X 0,Y 197.82,Z 909.018,A -85,B 0,C 180,E1 -21512.036,E2 -21512.036} C_VEL
LIN {X 0,Y 198.782,Z 905.289,A -85,B 0,C 180,E1 -21516.089,E2 -21516.089} C_VEL
LIN {X 0,Y 200.543,Z 900.037,A -85,B 0,C 180,E1 -21520.092,E2 -21520.092} C_VEL
LIN {X 0,Y 202.212,Z 894.986,A -85,B 0,C 180,E1 -21523.057,E2 -21523.057} C_VEL
LIN {X 0,Y 204.562,Z 887.78,A -85,B 0,C 180,E1 -21526.466,E2 -21526.466} C_VEL
LIN {X 0,Y 207.251,Z 880.212,A -85,B 0,C 180,E1 -21529.307,E2 -21529.307} C_VEL
LIN {X 0,Y 210.431,Z 871.127,A -85,B 0,C 180,E1 -21532.07,E2 -21532.07} C_VEL
LIN {X 0,Y 213.372,Z 862.07,A -85,B 0,C 180,E1 -21534.313,E2 -21534.313} C_VEL
LIN {X 0,Y 216.057,Z 852.451,A -85,B 0,C 180,E1 -21536.309,E2 -21536.309} C_VEL
LIN {X 0,Y 218.637,Z 842.307,A -85,B 0,C 180,E1 -21538.042,E2 -21538.042} C_VEL
LIN {X 0,Y 221.51,Z 829.914,A -85,B 0,C 180,E1 -21539.719,E2 -21539.719} C_VEL
LIN {X 0,Y 224.208,Z 816.049,A -85,B 0,C 180,E1 -21541.145,E2 -21541.145} C_VEL
LIN {X 0,Y 226.168,Z 802.066,A -85,B 0,C 180,E1 -21542.217,E2 -21542.217} C_VEL
LIN {X 0,Y 227.539,Z 787.264,A -85,B 0,C 180,E1 -21542.983,E2 -21542.983} C_VEL
LIN {X 0,Y 231.368,Z 714.156,A -85,B 0,C 180,E1 -21545.118,E2 -21545.118} C_VEL
LIN {X 0,Y 227.137,Z 704.514,A -85,B 0,C 180,E1 -21546.345,E2 -21546.345} C_VEL
LIN {X 0,Y 219.589,Z 690.555,A -85,B 0,C 180,E1 -21548.573,E2 -21548.573} C_VEL
LIN {X 0,Y 211.217,Z 677.134,A -85,B 0,C 180,E1 -21551.237,E2 -21551.237} C_VEL
LIN {X 0,Y 205.381,Z 668.812,A -85,B 0,C 180,E1 -21553.252,E2 -21553.252} C_VEL
LIN {X 0,Y 203.193,Z 665.631,A -85,B 0,C 180,E1 -21554.061,E2 -21554.061} C_VEL
LIN {X 0,Y 202.475,Z 664.616,A -85,B 0,C 180,E1 -21554.331,E2 -21554.331} C_VEL
LIN {X 0,Y 200.478,Z 662.403,A -85,B 0,C 180,E1 -21555.068,E2 -21555.068} C_VEL
LIN {X 0,Y 199.602,Z 659.748,A -85,B 0,C 180,E1 -21555.538,E2 -21555.538} C_VEL
LIN {X 0,Y 199.598,Z 659.721,A -85,B 0,C 180,E1 -21560.773,E2 -21560.773} C_VEL
LIN {X 0,Y 199.613,Z 659.735,A -85,B 0,C 180,E1 -21565.713,E2 -21565.713} C_VEL
LIN {X 0,Y 199.688,Z 659.728,A -85,B 0,C 180,E1 -21568.134,E2 -21568.134} C_VEL
LIN {X 0,Y 199.646,Z 659.742,A -85,B 0,C 180,E1 -21572.765,E2 -21572.765} C_VEL
LIN {X 0,Y 199.71,Z 659.718,A -85,B 0,C 180,E1 -21577.225,E2 -21577.225} C_VEL
LIN {X 0,Y 199.753,Z 659.704,A -85,B 0,C 180,E1 -21581.798,E2 -21581.798} C_VEL
LIN {X 0,Y 199.818,Z 659.72,A -85,B 0,C 180,E1 -21585.746,E2 -21585.746} C_VEL
LIN {X 0,Y 200.025,Z 659.668,A -85,B 0,C 180,E1 -21589.881,E2 -21589.881} C_VEL
LIN {X 0,Y 200.013,Z 659.694,A -85,B 0,C 180,E1 -21593.948,E2 -21593.948} C_VEL
LIN {X 0,Y 200.319,Z 659.657,A -85,B 0,C 180,E1 -21597.989,E2 -21597.989} C_VEL
LIN {X 0,Y 200.478,Z 659.629,A -85,B 0,C 180,E1 -21599.999,E2 -21599.999} C_VEL
LIN {X 0,Y 200.029,Z 659.692,A -85,B 0,C 180,E1 -21604.029,E2 -21604.029} C_VEL
LIN {X 0,Y 200.091,Z 659.686,A -85,B 0,C 180,E1 -21608.076,E2 -21608.076} C_VEL
LIN {X 0,Y 199.877,Z 659.707,A -85,B 0,C 180,E1 -21612.179,E2 -21612.179} C_VEL
LIN {X 0,Y 199.806,Z 659.712,A -85,B 0,C 180,E1 -21616.343,E2 -21616.343} C_VEL
LIN {X 0,Y 199.684,Z 659.727,A -85,B 0,C 180,E1 -21620.606,E2 -21620.606} C_VEL
LIN {X 0,Y 199.666,Z 659.734,A -85,B 0,C 180,E1 -21624.985,E2 -21624.985} C_VEL
LIN {X 0,Y 199.676,Z 659.737,A -85,B 0,C 180,E1 -21629.521,E2 -21629.521} C_VEL
LIN {X 0,Y 199.666,Z 659.739,A -85,B 0,C 180,E1 -21632.352,E2 -21632.352} C_VEL
LIN {X 0,Y 199.722,Z 659.833,A -85,B 0,C 180,E1 -21637.771,E2 -21637.771} C_VEL
LIN {X 0,Y 200.698,Z 662.833,A -85,B 0,C 180,E1 -21639.519,E2 -21639.519} C_VEL
LIN {X 0,Y 202.969,Z 666.681,A -85,B 0,C 180,E1 -21640.419,E2 -21640.419} C_VEL
LIN {X 0,Y 207.867,Z 674.578,A -85,B 0,C 180,E1 -21642.229,E2 -21642.229} C_VEL
LIN {X 0,Y 212.45,Z 682.555,A -85,B 0,C 180,E1 -21643.827,E2 -21643.827} C_VEL
LIN {X 0,Y 214.06,Z 685.488,A -85,B 0,C 180,E1 -21644.369,E2 -21644.369} C_VEL
LIN {X 0,Y 215.704,Z 690.626,A -85,B 0,C 180,E1 -21645.003,E2 -21645.003} C_VEL
LIN {X 0,Y 218.584,Z 707.697,A -85,B 0,C 180,E1 -21646.423,E2 -21646.423} C_VEL
LIN {X 0,Y 219.625,Z 711.309,A -85,B 0,C 180,E1 -21646.812,E2 -21646.812} C_VEL
LIN {X 0,Y 224.451,Z 724.085,A -85,B 0,C 180,E1 -21648.38,E2 -21648.38} C_VEL
LIN {X 0,Y 225.129,Z 730.924,A -85,B 0,C 180,E1 -21648.795,E2 -21648.795} C_VEL
LIN {X 0,Y 221.293,Z 802.091,A -85,B 0,C 180,E1 -21650.934,E2 -21650.934} C_VEL
LIN {X 0,Y 219.733,Z 815.935,A -85,B 0,C 180,E1 -21651.633,E2 -21651.633} C_VEL
LIN {X 0,Y 217.62,Z 828.969,A -85,B 0,C 180,E1 -21652.587,E2 -21652.587} C_VEL
LIN {X 0,Y 214.816,Z 842.339,A -85,B 0,C 180,E1 -21653.921,E2 -21653.921} C_VEL
LIN {X 0,Y 211.578,Z 855.214,A -85,B 0,C 180,E1 -21655.619,E2 -21655.619} C_VEL
LIN {X 0,Y 208.304,Z 867.105,A -85,B 0,C 180,E1 -21657.655,E2 -21657.655} C_VEL
LIN {X 0,Y 205.287,Z 876.679,A -85,B 0,C 180,E1 -21659.671,E2 -21659.671} C_VEL
LIN {X 0,Y 201.558,Z 887.472,A -85,B 0,C 180,E1 -21662.483,E2 -21662.483} C_VEL
LIN {X 0,Y 198.451,Z 896.389,A -85,B 0,C 180,E1 -21665.41,E2 -21665.41} C_VEL
LIN {X 0,Y 195.404,Z 904.93,A -85,B 0,C 180,E1 -21668.92,E2 -21668.92} C_VEL
LIN {X 0,Y 193.515,Z 910.901,A -85,B 0,C 180,E1 -21672.019,E2 -21672.019} C_VEL
LIN {X 0,Y 192.008,Z 915.823,A -85,B 0,C 180,E1 -21675.154,E2 -21675.154} C_VEL
LIN {X 0,Y 190.76,Z 920.906,A -85,B 0,C 180,E1 -21679.385,E2 -21679.385} C_VEL
LIN {X 0,Y 190.3,Z 924.468,A -85,B 0,C 180,E1 -21683.639,E2 -21683.639} C_VEL
LIN {X 0,Y 190.265,Z 926.604,A -85,B 0,C 180,E1 -21687.883,E2 -21687.883} C_VEL
LIN {X 0,Y 190.39,Z 927.157,A -85,B 0,C 180,E1 -21690,E2 -21690} C_VEL
LIN {X 0,Y 190.194,Z 927.223,A -85,B 0,C 180,E1 -21694.238,E2 -21694.238} C_VEL
LIN {X 0,Y 190.438,Z 925.954,A -85,B 0,C 180,E1 -21698.489,E2 -21698.489} C_VEL
LIN {X 0,Y 191.334,Z 923.331,A -85,B 0,C 180,E1 -21702.732,E2 -21702.732} C_VEL
LIN {X 0,Y 193.215,Z 919.279,A -85,B 0,C 180,E1 -21706.917,E2 -21706.917} C_VEL
LIN {X 0,Y 195.896,Z 913.685,A -85,B 0,C 180,E1 -21711.024,E2 -21711.024} C_VEL
LIN {X 0,Y 198.986,Z 907.403,A -85,B 0,C 180,E1 -21714.519,E2 -21714.519} C_VEL
LIN {X 0,Y 202.921,Z 899.605,A -85,B 0,C 180,E1 -21717.876,E2 -21717.876} C_VEL
LIN {X 0,Y 206.84,Z 891.487,A -85,B 0,C 180,E1 -21720.642,E2 -21720.642} C_VEL
LIN {X 0,Y 211.269,Z 881.725,A -85,B 0,C 180,E1 -21723.29,E2 -21723.29} C_VEL
LIN {X 0,Y 215.534,Z 871.074,A -85,B 0,C 180,E1 -21725.607,E2 -21725.607} C_VEL
LIN {X 0,Y 219.946,Z 858.944,A -85,B 0,C 180,E1 -21727.669,E2 -21727.669} C_VEL
LIN {X 0,Y 223.726,Z 847.175,A -85,B 0,C 180,E1 -21729.212,E2 -21729.212} C_VEL
LIN {X 0,Y 227.126,Z 834.325,A -85,B 0,C 180,E1 -21730.527,E2 -21730.527} C_VEL
LIN {X 0,Y 229.885,Z 821.195,A -85,B 0,C 180,E1 -21731.531,E2 -21731.531} C_VEL
LIN {X 0,Y 232.14,Z 806.695,A -85,B 0,C 180,E1 -21732.291,E2 -21732.291} C_VEL
LIN {X 0,Y 233.506,Z 790.56,A -85,B 0,C 180,E1 -21732.833,E2 -21732.833} C_VEL
LIN {X 0,Y 236.776,Z 736.267,A -85,B 0,C 180,E1 -21734.343,E2 -21734.343} C_VEL
LIN {X 0,Y 232.121,Z 724.852,A -85,B 0,C 180,E1 -21736.077,E2 -21736.077} C_VEL
LIN {X 0,Y 226.32,Z 712.527,A -85,B 0,C 180,E1 -21738.337,E2 -21738.337} C_VEL
LIN {X 0,Y 219.8,Z 700.265,A -85,B 0,C 180,E1 -21741.087,E2 -21741.087} C_VEL
LIN {X 0,Y 213.729,Z 690.152,A -85,B 0,C 180,E1 -21743.906,E2 -21743.906} C_VEL
LIN {X 0,Y 209.928,Z 684.3,A -85,B 0,C 180,E1 -21745.841,E2 -21745.841} C_VEL
LIN {X 0,Y 206.332,Z 678.907,A -85,B 0,C 180,E1 -21747.837,E2 -21747.837} C_VEL
LIN {X 0,Y 203.164,Z 674.333,A -85,B 0,C 180,E1 -21749.753,E2 -21749.753} C_VEL
LIN {X 0,Y 198.237,Z 668.19,A -85,B 0,C 180,E1 -21753.056,E2 -21753.056} C_VEL
LIN {X 0,Y 197.246,Z 666.443,A -85,B 0,C 180,E1 -21753.837,E2 -21753.837} C_VEL
LIN {X 0,Y 194.536,Z 664.585,A -85,B 0,C 180,E1 -21755.872,E2 -21755.872} C_VEL
LIN {X 0,Y 193.051,Z 662.107,A -85,B 0,C 180,E1 -21757.245,E2 -21757.245} C_VEL
LIN {X 0,Y 192.681,Z 660.595,A -85,B 0,C 180,E1 -21757.764,E2 -21757.764} C_VEL
LIN {X 0,Y 192.759,Z 660.591,A -85,B 0,C 180,E1 -21763.042,E2 -21763.042} C_VEL
LIN {X 0,Y 192.806,Z 660.583,A -85,B 0,C 180,E1 -21767.367,E2 -21767.367} C_VEL
LIN {X 0,Y 193.042,Z 660.55,A -85,B 0,C 180,E1 -21771.627,E2 -21771.627} C_VEL
LIN {X 0,Y 193.264,Z 660.536,A -85,B 0,C 180,E1 -21777.917,E2 -21777.917} C_VEL
LIN {X 0,Y 193.442,Z 660.5,A -85,B 0,C 180,E1 -21780.001,E2 -21780.001} C_VEL
LIN {X 0,Y 192.975,Z 660.563,A -85,B 0,C 180,E1 -21784.178,E2 -21784.178} C_VEL
LIN {X 0,Y 193.038,Z 660.564,A -85,B 0,C 180,E1 -21788.374,E2 -21788.374} C_VEL
LIN {X 0,Y 192.804,Z 660.594,A -85,B 0,C 180,E1 -21792.634,E2 -21792.634} C_VEL
LIN {X 0,Y 192.787,Z 660.784,A -85,B 0,C 180,E1 -21797.984,E2 -21797.984} C_VEL
LIN {X 0,Y 193.571,Z 663.223,A -85,B 0,C 180,E1 -21798.851,E2 -21798.851} C_VEL
LIN {X 0,Y 195.393,Z 665.374,A -85,B 0,C 180,E1 -21800.393,E2 -21800.393} C_VEL
LIN {X 0,Y 197.528,Z 666.615,A -85,B 0,C 180,E1 -21801.938,E2 -21801.938} C_VEL
LIN {X 0,Y 199.118,Z 669.581,A -85,B 0,C 180,E1 -21803.179,E2 -21803.179} C_VEL
LIN {X 0,Y 201.705,Z 671.88,A -85,B 0,C 180,E1 -21804.854,E2 -21804.854} C_VEL
LIN {X 0,Y 202.486,Z 673.049,A -85,B 0,C 180,E1 -21805.369,E2 -21805.369} C_VEL
LIN {X 0,Y 204.959,Z 676.273,A -85,B 0,C 180,E1 -21806.886,E2 -21806.886} C_VEL
LIN {X 0,Y 206.375,Z 677.725,A -85,B 0,C 180,E1 -21807.681,E2 -21807.681} C_VEL
LIN {X 0,Y 209.133,Z 681.395,A -85,B 0,C 180,E1 -21809.201,E2 -21809.201} C_VEL
LIN {X 0,Y 210.461,Z 683.17,A -85,B 0,C 180,E1 -21809.896,E2 -21809.896} C_VEL
LIN {X 0,Y 214.318,Z 688.356,A -85,B 0,C 180,E1 -21811.799,E2 -21811.799} C_VEL
LIN {X 0,Y 219.069,Z 694.938,A -85,B 0,C 180,E1 -21813.947,E2 -21813.947} C_VEL
LIN {X 0,Y 226.339,Z 706.132,A -85,B 0,C 180,E1 -21816.933,E2 -21816.933} C_VEL
LIN {X 0,Y 233.18,Z 717.915,A -85,B 0,C 180,E1 -21819.477,E2 -21819.477} C_VEL
LIN {X 0,Y 237.04,Z 725.911,A -85,B 0,C 180,E1 -21820.854,E2 -21820.854} C_VEL
LIN {X 0,Y 237.288,Z 726.487,A -85,B 0,C 180,E1 -21820.943,E2 -21820.943} C_VEL
LIN {X 0,Y 233.434,Z 788.911,A -85,B 0,C 180,E1 -21822.725,E2 -21822.725} C_VEL
LIN {X 0,Y 231.642,Z 803.378,A -85,B 0,C 180,E1 -21823.426,E2 -21823.426} C_VEL
LIN {X 0,Y 229.274,Z 816.818,A -85,B 0,C 180,E1 -21824.389,E2 -21824.389} C_VEL
LIN {X 0,Y 225.96,Z 830.427,A -85,B 0,C 180,E1 -21825.674,E2 -21825.674} C_VEL
LIN {X 0,Y 222.532,Z 842.613,A -85,B 0,C 180,E1 -21827.234,E2 -21827.234} C_VEL
LIN {X 0,Y 218.594,Z 854.127,A -85,B 0,C 180,E1 -21829.075,E2 -21829.075} C_VEL
LIN {X 0,Y 214.142,Z 865.652,A -85,B 0,C 180,E1 -21831.423,E2 -21831.423} C_VEL
LIN {X 0,Y 210.493,Z 874.306,A -85,B 0,C 180,E1 -21833.655,E2 -21833.655} C_VEL
LIN {X 0,Y 206.374,Z 883.034,A -85,B 0,C 180,E1 -21836.4,E2 -21836.4} C_VEL
LIN {X 0,Y 202.159,Z 891.377,A -85,B 0,C 180,E1 -21839.729,E2 -21839.729} C_VEL
LIN {X 0,Y 199.093,Z 897.159,A -85,B 0,C 180,E1 -21842.684,E2 -21842.684} C_VEL
LIN {X 0,Y 196.476,Z 901.904,A -85,B 0,C 180,E1 -21845.71,E2 -21845.71} C_VEL
LIN {X 0,Y 193.791,Z 906.789,A -85,B 0,C 180,E1 -21849.847,E2 -21849.847} C_VEL
LIN {X 0,Y 192.279,Z 909.45,A -85,B 0,C 180,E1 -21852.998,E2 -21852.998} C_VEL
LIN {X 0,Y 190.91,Z 911.752,A -85,B 0,C 180,E1 -21857.24,E2 -21857.24} C_VEL
LIN {X 0,Y 190.392,Z 912.704,A -85,B 0,C 180,E1 -21861.509,E2 -21861.509} C_VEL
LIN {X 0,Y 190.318,Z 912.346,A -85,B 0,C 180,E1 -21865.765,E2 -21865.765} C_VEL
LIN {X 0,Y 190.496,Z 910.687,A -85,B 0,C 180,E1 -21870,E2 -21870} C_VEL
LIN {X 0,Y 191.14,Z 907.69,A -85,B 0,C 180,E1 -21874.217,E2 -21874.217} C_VEL
LIN {X 0,Y 192.585,Z 903.261,A -85,B 0,C 180,E1 -21878.394,E2 -21878.394} C_VEL
LIN {X 0,Y 194.117,Z 898.867,A -85,B 0,C 180,E1 -21881.486,E2 -21881.486} C_VEL
LIN {X 0,Y 196.017,Z 893.529,A -85,B 0,C 180,E1 -21884.536,E2 -21884.536} C_VEL
LIN {X 0,Y 198.587,Z 885.899,A -85,B 0,C 180,E1 -21888.039,E2 -21888.039} C_VEL
LIN {X 0,Y 201.7,Z 877.903,A -85,B 0,C 180,E1 -21890.925,E2 -21890.925} C_VEL
LIN {X 0,Y 205.098,Z 868.279,A -85,B 0,C 180,E1 -21893.743,E2 -21893.743} C_VEL
LIN {X 0,Y 208.394,Z 857.621,A -85,B 0,C 180,E1 -21896.272,E2 -21896.272} C_VEL
LIN {X 0,Y 211.32,Z 847.096,A -85,B 0,C 180,E1 -21898.289,E2 -21898.289} C_VEL
LIN {X 0,Y 214.683,Z 834.189,A -85,B 0,C 180,E1 -21900.221,E2 -21900.221} C_VEL
LIN {X 0,Y 217.422,Z 821.516,A -85,B 0,C 180,E1 -21901.687,E2 -21901.687} C_VEL
LIN {X 0,Y 219.737,Z 807.277,A -85,B 0,C 180,E1 -21902.938,E2 -21902.938} C_VEL
LIN {X 0,Y 221.397,Z 792.736,A -85,B 0,C 180,E1 -21903.815,E2 -21903.815} C_VEL
LIN {X 0,Y 222.529,Z 775.495,A -85,B 0,C 180,E1 -21904.439,E2 -21904.439} C_VEL
LIN {X 0,Y 225.754,Z 716.368,A -85,B 0,C 180,E1 -21906.155,E2 -21906.155} C_VEL
LIN {X 0,Y 222.371,Z 708.618,A -85,B 0,C 180,E1 -21907.188,E2 -21907.188} C_VEL
LIN {X 0,Y 214.926,Z 694.687,A -85,B 0,C 180,E1 -21909.499,E2 -21909.499} C_VEL
LIN {X 0,Y 207.096,Z 681.982,A -85,B 0,C 180,E1 -21912.122,E2 -21912.122} C_VEL
LIN {X 0,Y 201.289,Z 673.7,A -85,B 0,C 180,E1 -21914.228,E2 -21914.228} C_VEL
LIN {X 0,Y 198.823,Z 670.115,A -85,B 0,C 180,E1 -21915.189,E2 -21915.189} C_VEL
LIN {X 0,Y 196.601,Z 667.225,A -85,B 0,C 180,E1 -21916.073,E2 -21916.073} C_VEL
LIN {X 0,Y 195.704,Z 665.703,A -85,B 0,C 180,E1 -21916.46,E2 -21916.46} C_VEL
LIN {X 0,Y 193.524,Z 663.485,A -85,B 0,C 180,E1 -21917.344,E2 -21917.344} C_VEL
LIN {X 0,Y 192.568,Z 660.842,A -85,B 0,C 180,E1 -21917.84,E2 -21917.84} C_VEL
LIN {X 0,Y 192.546,Z 660.621,A -85,B 0,C 180,E1 -21918.008,E2 -21918.008} C_VEL
LIN {X 0,Y 192.582,Z 660.58,A -85,B 0,C 180,E1 -21923.404,E2 -21923.404} C_VEL
LIN {X 0,Y 192.608,Z 660.62,A -85,B 0,C 180,E1 -21927.061,E2 -21927.061} C_VEL
LIN {X 0,Y 192.623,Z 660.609,A -85,B 0,C 180,E1 -21931.684,E2 -21931.684} C_VEL
LIN {X 0,Y 192.681,Z 660.587,A -85,B 0,C 180,E1 -21936.345,E2 -21936.345} C_VEL
LIN {X 0,Y 192.701,Z 660.584,A -85,B 0,C 180,E1 -21941.487,E2 -21941.487} C_VEL
LIN {X 0,Y 192.743,Z 660.598,A -85,B 0,C 180,E1 -21945.211,E2 -21945.211} C_VEL
LIN {X 0,Y 192.948,Z 660.549,A -85,B 0,C 180,E1 -21949.566,E2 -21949.566} C_VEL
LIN {X 0,Y 192.976,Z 660.572,A -85,B 0,C 180,E1 -21953.727,E2 -21953.727} C_VEL
LIN {X 0,Y 193.26,Z 660.536,A -85,B 0,C 180,E1 -21957.915,E2 -21957.915} C_VEL
LIN {X 0,Y 193.442,Z 660.505,A -85,B 0,C 180,E1 -21959.999,E2 -21959.999} C_VEL
LIN {X 0,Y 192.975,Z 660.57,A -85,B 0,C 180,E1 -21964.176,E2 -21964.176} C_VEL
LIN {X 0,Y 193.039,Z 660.565,A -85,B 0,C 180,E1 -21968.373,E2 -21968.373} C_VEL
LIN {X 0,Y 192.804,Z 660.593,A -85,B 0,C 180,E1 -21972.633,E2 -21972.633} C_VEL
LIN {X 0,Y 192.759,Z 660.595,A -85,B 0,C 180,E1 -21976.958,E2 -21976.958} C_VEL
LIN {X 0,Y 192.619,Z 660.613,A -85,B 0,C 180,E1 -21981.399,E2 -21981.399} C_VEL
LIN {X 0,Y 192.649,Z 660.602,A -85,B 0,C 180,E1 -21984.213,E2 -21984.213} C_VEL
LIN {X 0,Y 192.651,Z 660.611,A -85,B 0,C 180,E1 -21988.892,E2 -21988.892} C_VEL
LIN {X 0,Y 192.601,Z 660.616,A -85,B 0,C 180,E1 -21993.185,E2 -21993.185} C_VEL
LIN {X 0,Y 192.632,Z 660.742,A -85,B 0,C 180,E1 -21995.98,E2 -21995.98} C_VEL
LIN {X 0,Y 193.024,Z 662.205,A -85,B 0,C 180,E1 -21996.898,E2 -21996.898} C_VEL
LIN {X 0,Y 195.826,Z 666.573,A -85,B 0,C 180,E1 -21998.124,E2 -21998.124} C_VEL
LIN {X 0,Y 197.284,Z 668.723,A -85,B 0,C 180,E1 -21998.73,E2 -21998.73} C_VEL
LIN {X 0,Y 201.245,Z 675.153,A -85,B 0,C 180,E1 -22000.327,E2 -22000.327} C_VEL
LIN {X 0,Y 206.248,Z 683.649,A -85,B 0,C 180,E1 -22002.215,E2 -22002.215} C_VEL
LIN {X 0,Y 213.623,Z 697.731,A -85,B 0,C 180,E1 -22004.81,E2 -22004.81} C_VEL
LIN {X 0,Y 219.625,Z 711.309,A -85,B 0,C 180,E1 -22006.812,E2 -22006.812} C_VEL
LIN {X 0,Y 220.425,Z 714.951,A -85,B 0,C 180,E1 -22007.143,E2 -22007.143} C_VEL
LIN {X 0,Y 220.445,Z 721.492,A -85,B 0,C 180,E1 -22007.421,E2 -22007.421} C_VEL
LIN {X 0,Y 219.562,Z 732.346,A -85,B 0,C 180,E1 -22007.681,E2 -22007.681} C_VEL
LIN {X 0,Y 215.679,Z 801.51,A -85,B 0,C 180,E1 -22009.789,E2 -22009.789} C_VEL
LIN {X 0,Y 214.085,Z 815.464,A -85,B 0,C 180,E1 -22010.502,E2 -22010.502} C_VEL
LIN {X 0,Y 211.964,Z 827.973,A -85,B 0,C 180,E1 -22011.409,E2 -22011.409} C_VEL
LIN {X 0,Y 209.111,Z 841.508,A -85,B 0,C 180,E1 -22012.774,E2 -22012.774} C_VEL
LIN {X 0,Y 205.742,Z 854.49,A -85,B 0,C 180,E1 -22014.499,E2 -22014.499} C_VEL
LIN {X 0,Y 202.458,Z 865.732,A -85,B 0,C 180,E1 -22016.42,E2 -22016.42} C_VEL
LIN {X 0,Y 199.09,Z 876.089,A -85,B 0,C 180,E1 -22018.622,E2 -22018.622} C_VEL
LIN {X 0,Y 195.853,Z 885.294,A -85,B 0,C 180,E1 -22021.024,E2 -22021.024} C_VEL
LIN {X 0,Y 192.471,Z 894.528,A -85,B 0,C 180,E1 -22024.012,E2 -22024.012} C_VEL
LIN {X 0,Y 189.183,Z 903.35,A -85,B 0,C 180,E1 -22027.618,E2 -22027.618} C_VEL
LIN {X 0,Y 187.295,Z 908.633,A -85,B 0,C 180,E1 -22030.262,E2 -22030.262} C_VEL
LIN {X 0,Y 185.594,Z 913.9,A -85,B 0,C 180,E1 -22033.5,E2 -22033.5} C_VEL
LIN {X 0,Y 183.971,Z 919.448,A -85,B 0,C 180,E1 -22037.871,E2 -22037.871} C_VEL
LIN {X 0,Y 183.384,Z 922.524,A -85,B 0,C 180,E1 -22041.182,E2 -22041.182} C_VEL
LIN {X 0,Y 183.152,Z 925.393,A -85,B 0,C 180,E1 -22045.598,E2 -22045.598} C_VEL
LIN {X 0,Y 183.309,Z 926.866,A -85,B 0,C 180,E1 -22050,E2 -22050} C_VEL
LIN {X 0,Y 183.114,Z 926.956,A -85,B 0,C 180,E1 -22054.402,E2 -22054.402} C_VEL
LIN {X 0,Y 183.385,Z 925.711,A -85,B 0,C 180,E1 -22058.818,E2 -22058.818} C_VEL
LIN {X 0,Y 184.359,Z 923.119,A -85,B 0,C 180,E1 -22063.222,E2 -22063.222} C_VEL
LIN {X 0,Y 186.379,Z 919.102,A -85,B 0,C 180,E1 -22067.557,E2 -22067.557} C_VEL
LIN {X 0,Y 189.159,Z 913.63,A -85,B 0,C 180,E1 -22071.745,E2 -22071.745} C_VEL
LIN {X 0,Y 192.515,Z 907.287,A -85,B 0,C 180,E1 -22075.401,E2 -22075.401} C_VEL
LIN {X 0,Y 196.617,Z 899.524,A -85,B 0,C 180,E1 -22078.852,E2 -22078.852} C_VEL
LIN {X 0,Y 200.747,Z 891.447,A -85,B 0,C 180,E1 -22081.678,E2 -22081.678} C_VEL
LIN {X 0,Y 205.348,Z 881.734,A -85,B 0,C 180,E1 -22084.382,E2 -22084.382} C_VEL
LIN {X 0,Y 209.846,Z 871.017,A -85,B 0,C 180,E1 -22086.762,E2 -22086.762} C_VEL
LIN {X 0,Y 214.387,Z 859.082,A -85,B 0,C 180,E1 -22088.826,E2 -22088.826} C_VEL
LIN {X 0,Y 218.28,Z 847.407,A -85,B 0,C 180,E1 -22090.388,E2 -22090.388} C_VEL
LIN {X 0,Y 222.033,Z 833.691,A -85,B 0,C 180,E1 -22091.812,E2 -22091.812} C_VEL
LIN {X 0,Y 225.054,Z 819.666,A -85,B 0,C 180,E1 -22092.858,E2 -22092.858} C_VEL
LIN {X 0,Y 227.209,Z 805.498,A -85,B 0,C 180,E1 -22093.593,E2 -22093.593} C_VEL
LIN {X 0,Y 228.693,Z 787.94,A -85,B 0,C 180,E1 -22094.161,E2 -22094.161} C_VEL
LIN {X 0,Y 231.783,Z 738.598,A -85,B 0,C 180,E1 -22095.548,E2 -22095.548} C_VEL
LIN {X 0,Y 227.346,Z 727.652,A -85,B 0,C 180,E1 -22097.302,E2 -22097.302} C_VEL
LIN {X 0,Y 222.057,Z 716.271,A -85,B 0,C 180,E1 -22099.494,E2 -22099.494} C_VEL
LIN {X 0,Y 216.133,Z 705.003,A -85,B 0,C 180,E1 -22102.139,E2 -22102.139} C_VEL
LIN {X 0,Y 210.591,Z 695.535,A -85,B 0,C 180,E1 -22104.86,E2 -22104.86} C_VEL
LIN {X 0,Y 207.036,Z 689.875,A -85,B 0,C 180,E1 -22106.773,E2 -22106.773} C_VEL
LIN {X 0,Y 203.663,Z 684.727,A -85,B 0,C 180,E1 -22108.744,E2 -22108.744} C_VEL
LIN {X 0,Y 200.04,Z 679.445,A -85,B 0,C 180,E1 -22111.072,E2 -22111.072} C_VEL
LIN {X 0,Y 196.109,Z 674.314,A -85,B 0,C 180,E1 -22113.888,E2 -22113.888} C_VEL
LIN {X 0,Y 195.447,Z 673.099,A -85,B 0,C 180,E1 -22114.438,E2 -22114.438} C_VEL
LIN {X 0,Y 192.818,Z 671.131,A -85,B 0,C 180,E1 -22116.506,E2 -22116.506} C_VEL
LIN {X 0,Y 191.136,Z 668.287,A -85,B 0,C 180,E1 -22118.143,E2 -22118.143} C_VEL
LIN {X 0,Y 190.791,Z 667.449,A -85,B 0,C 180,E1 -22118.528,E2 -22118.528} C_VEL
LIN {X 0,Y 188.145,Z 666.03,A -85,B 0,C 180,E1 -22121.158,E2 -22121.158} C_VEL
LIN {X 0,Y 186.282,Z 663.551,A -85,B 0,C 180,E1 -22123.564,E2 -22123.564} C_VEL
LIN {X 0,Y 185.714,Z 661.471,A -85,B 0,C 180,E1 -22124.71,E2 -22124.71} C_VEL
LIN {X 0,Y 185.889,Z 661.447,A -85,B 0,C 180,E1 -22129.418,E2 -22129.418} C_VEL
LIN {X 0,Y 185.953,Z 661.448,A -85,B 0,C 180,E1 -22133.49,E2 -22133.49} C_VEL
LIN {X 0,Y 186.208,Z 661.414,A -85,B 0,C 180,E1 -22137.838,E2 -22137.838} C_VEL
LIN {X 0,Y 186.406,Z 661.376,A -85,B 0,C 180,E1 -22140.001,E2 -22140.001} C_VEL
LIN {X 0,Y 185.922,Z 661.44,A -85,B 0,C 180,E1 -22144.336,E2 -22144.336} C_VEL
LIN {X 0,Y 185.985,Z 661.438,A -85,B 0,C 180,E1 -22148.694,E2 -22148.694} C_VEL
LIN {X 0,Y 185.856,Z 661.593,A -85,B 0,C 180,E1 -22151.175,E2 -22151.175} C_VEL
LIN {X 0,Y 186.448,Z 663.742,A -85,B 0,C 180,E1 -22152.242,E2 -22152.242} C_VEL
LIN {X 0,Y 188.074,Z 665.926,A -85,B 0,C 180,E1 -22154.334,E2 -22154.334} C_VEL
LIN {X 0,Y 190.953,Z 667.624,A -85,B 0,C 180,E1 -22157.207,E2 -22157.207} C_VEL
LIN {X 0,Y 192.235,Z 670.394,A -85,B 0,C 180,E1 -22158.548,E2 -22158.548} C_VEL
LIN {X 0,Y 194.815,Z 672.797,A -85,B 0,C 180,E1 -22160.68,E2 -22160.68} C_VEL
LIN {X 0,Y 195.673,Z 673.47,A -85,B 0,C 180,E1 -22161.326,E2 -22161.326} C_VEL
LIN {X 0,Y 197.841,Z 676.833,A -85,B 0,C 180,E1 -22163.002,E2 -22163.002} C_VEL
LIN {X 0,Y 200.046,Z 678.923,A -85,B 0,C 180,E1 -22164.469,E2 -22164.469} C_VEL
LIN {X 0,Y 202.717,Z 682.542,A -85,B 0,C 180,E1 -22166.192,E2 -22166.192} C_VEL
LIN {X 0,Y 204.191,Z 684.257,A -85,B 0,C 180,E1 -22167.064,E2 -22167.064} C_VEL
LIN {X 0,Y 207.884,Z 689.221,A -85,B 0,C 180,E1 -22169.147,E2 -22169.147} C_VEL
LIN {X 0,Y 211.38,Z 694.002,A -85,B 0,C 180,E1 -22170.952,E2 -22170.952} C_VEL
LIN {X 0,Y 216.03,Z 700.624,A -85,B 0,C 180,E1 -22173.156,E2 -22173.156} C_VEL
LIN {X 0,Y 223.266,Z 712.055,A -85,B 0,C 180,E1 -22176.26,E2 -22176.26} C_VEL
LIN {X 0,Y 230.087,Z 724.18,A -85,B 0,C 180,E1 -22178.902,E2 -22178.902} C_VEL
LIN {X 0,Y 232.285,Z 728.912,A -85,B 0,C 180,E1 -22179.73,E2 -22179.73} C_VEL
LIN {X 0,Y 228.445,Z 789.185,A -85,B 0,C 180,E1 -22181.479,E2 -22181.479} C_VEL
LIN {X 0,Y 226.659,Z 803.258,A -85,B 0,C 180,E1 -22182.161,E2 -22182.161} C_VEL
LIN {X 0,Y 224.085,Z 817.37,A -85,B 0,C 180,E1 -22183.181,E2 -22183.181} C_VEL
LIN {X 0,Y 220.955,Z 829.796,A -85,B 0,C 180,E1 -22184.35,E2 -22184.35} C_VEL
LIN {X 0,Y 217.324,Z 842.344,A -85,B 0,C 180,E1 -22185.95,E2 -22185.95} C_VEL
LIN {X 0,Y 213.233,Z 853.954,A -85,B 0,C 180,E1 -22187.814,E2 -22187.814} C_VEL
LIN {X 0,Y 208.563,Z 865.554,A -85,B 0,C 180,E1 -22190.19,E2 -22190.19} C_VEL
LIN {X 0,Y 204.729,Z 874.27,A -85,B 0,C 180,E1 -22192.459,E2 -22192.459} C_VEL
LIN {X 0,Y 200.424,Z 883.049,A -85,B 0,C 180,E1 -22195.263,E2 -22195.263} C_VEL
LIN {X 0,Y 195.963,Z 891.441,A -85,B 0,C 180,E1 -22198.666,E2 -22198.666} C_VEL
LIN {X 0,Y 192.714,Z 897.261,A -85,B 0,C 180,E1 -22201.7,E2 -22201.7} C_VEL
LIN {X 0,Y 189.13,Z 903.456,A -85,B 0,C 180,E1 -22205.873,E2 -22205.873} C_VEL
LIN {X 0,Y 186.488,Z 907.964,A -85,B 0,C 180,E1 -22210.174,E2 -22210.174} C_VEL
LIN {X 0,Y 184.575,Z 910.994,A -85,B 0,C 180,E1 -22214.542,E2 -22214.542} C_VEL
LIN {X 0,Y 183.53,Z 912.646,A -85,B 0,C 180,E1 -22218.962,E2 -22218.962} C_VEL
LIN {X 0,Y 183.212,Z 912.97,A -85,B 0,C 180,E1 -22223.392,E2 -22223.392} C_VEL
LIN {X 0,Y 183.231,Z 912.606,A -85,B 0,C 180,E1 -22225.764,E2 -22225.764} C_VEL
LIN {X 0,Y 183.41,Z 911.013,A -85,B 0,C 180,E1 -22230,E2 -22230} C_VEL
LIN {X 0,Y 184.076,Z 908.048,A -85,B 0,C 180,E1 -22234.38,E2 -22234.38} C_VEL
LIN {X 0,Y 185.582,Z 903.651,A -85,B 0,C 180,E1 -22238.713,E2 -22238.713} C_VEL
LIN {X 0,Y 187.182,Z 899.294,A -85,B 0,C 180,E1 -22241.918,E2 -22241.918} C_VEL
LIN {X 0,Y 189.174,Z 893.994,A -85,B 0,C 180,E1 -22245.074,E2 -22245.074} C_VEL
LIN {X 0,Y 191.881,Z 886.405,A -85,B 0,C 180,E1 -22248.693,E2 -22248.693} C_VEL
LIN {X 0,Y 195.643,Z 876.988,A -85,B 0,C 180,E1 -22252.16,E2 -22252.16} C_VEL
LIN {X 0,Y 199.307,Z 867.121,A -85,B 0,C 180,E1 -22255.034,E2 -22255.034} C_VEL
LIN {X 0,Y 202.819,Z 856.175,A -85,B 0,C 180,E1 -22257.611,E2 -22257.611} C_VEL
LIN {X 0,Y 206.295,Z 843.935,A -85,B 0,C 180,E1 -22259.884,E2 -22259.884} C_VEL
LIN {X 0,Y 209.383,Z 831.799,A -85,B 0,C 180,E1 -22261.632,E2 -22261.632} C_VEL
LIN {X 0,Y 212.087,Z 819.426,A -85,B 0,C 180,E1 -22263.004,E2 -22263.004} C_VEL
LIN {X 0,Y 214.252,Z 805.687,A -85,B 0,C 180,E1 -22264.177,E2 -22264.177} C_VEL
LIN {X 0,Y 215.912,Z 791.338,A -85,B 0,C 180,E1 -22265.009,E2 -22265.009} C_VEL
LIN {X 0,Y 217.182,Z 770.542,A -85,B 0,C 180,E1 -22265.732,E2 -22265.732} C_VEL
LIN {X 0,Y 220.167,Z 718.469,A -85,B 0,C 180,E1 -22267.26,E2 -22267.26} C_VEL
LIN {X 0,Y 216.848,Z 711.117,A -85,B 0,C 180,E1 -22268.323,E2 -22268.323} C_VEL
LIN {X 0,Y 209.521,Z 697.348,A -85,B 0,C 180,E1 -22270.743,E2 -22270.743} C_VEL
LIN {X 0,Y 201.244,Z 684.091,A -85,B 0,C 180,E1 -22273.71,E2 -22273.71} C_VEL
LIN {X 0,Y 195.036,Z 675.337,A -85,B 0,C 180,E1 -22276.156,E2 -22276.156} C_VEL
LIN {X 0,Y 192.083,Z 671.228,A -85,B 0,C 180,E1 -22277.417,E2 -22277.417} C_VEL
LIN {X 0,Y 189.8,Z 668.34,A -85,B 0,C 180,E1 -22278.426,E2 -22278.426} C_VEL
LIN {X 0,Y 188.905,Z 666.74,A -85,B 0,C 180,E1 -22278.864,E2 -22278.864} C_VEL
LIN {X 0,Y 186.801,Z 664.807,A -85,B 0,C 180,E1 -22279.81,E2 -22279.81} C_VEL
LIN {X 0,Y 185.603,Z 662.281,A -85,B 0,C 180,E1 -22280.459,E2 -22280.459} C_VEL
LIN {X 0,Y 185.475,Z 661.48,A -85,B 0,C 180,E1 -22280.602,E2 -22280.602} C_VEL
LIN {X 0,Y 185.498,Z 661.483,A -85,B 0,C 180,E1 -22285.367,E2 -22285.367} C_VEL
LIN {X 0,Y 185.546,Z 661.48,A -85,B 0,C 180,E1 -22290.5,E2 -22290.5} C_VEL
LIN {X 0,Y 185.583,Z 661.471,A -85,B 0,C 180,E1 -22295.381,E2 -22295.381} C_VEL
LIN {X 0,Y 185.636,Z 661.467,A -85,B 0,C 180,E1 -22301.17,E2 -22301.17} C_VEL
LIN {X 0,Y 185.672,Z 661.471,A -85,B 0,C 180,E1 -22304.635,E2 -22304.635} C_VEL
LIN {X 0,Y 185.89,Z 661.428,A -85,B 0,C 180,E1 -22309.418,E2 -22309.418} C_VEL
LIN {X 0,Y 185.94,Z 661.45,A -85,B 0,C 180,E1 -22313.488,E2 -22313.488} C_VEL
LIN {X 0,Y 186.204,Z 661.414,A -85,B 0,C 180,E1 -22317.836,E2 -22317.836} C_VEL
LIN {X 0,Y 186.406,Z 661.381,A -85,B 0,C 180,E1 -22319.999,E2 -22319.999} C_VEL
LIN {X 0,Y 185.921,Z 661.448,A -85,B 0,C 180,E1 -22324.335,E2 -22324.335} C_VEL
LIN {X 0,Y 185.985,Z 661.443,A -85,B 0,C 180,E1 -22328.693,E2 -22328.693} C_VEL
LIN {X 0,Y 185.731,Z 661.474,A -85,B 0,C 180,E1 -22333.122,E2 -22333.122} C_VEL
LIN {X 0,Y 185.691,Z 661.477,A -85,B 0,C 180,E1 -22337.624,E2 -22337.624} C_VEL
LIN {X 0,Y 185.58,Z 661.488,A -85,B 0,C 180,E1 -22342.253,E2 -22342.253} C_VEL
LIN {X 0,Y 185.562,Z 661.486,A -85,B 0,C 180,E1 -22347.032,E2 -22347.032} C_VEL
LIN {X 0,Y 185.58,Z 661.493,A -85,B 0,C 180,E1 -22349.492,E2 -22349.492} C_VEL
LIN {X 0,Y 185.55,Z 661.544,A -85,B 0,C 180,E1 -22353.912,E2 -22353.912} C_VEL
